REGION Network 15: Start dosilanie minuty
   RUNG wire#powerrail
      "Detection_Changes_Data_Word_USInt"("tempdbHold_SendingTCP.sterowanie." := "tempdbHold_SendingTCP".Start_dosilanie_1.MINUTE, "DB10_instance_SCADA." := "DB10_instance_SCADA".actDTL_RechargingOn.MINUTE, memRisingTriger_Data_ := "memRisingTriger_Data_14", "dbHold_Sending.data.stat.control." := "dbHold_Sending".data."Time".Start_dosilanie_1.MINUTE)
      "Saving_Canged_Data_Word_USInt"("dbHold_download.sterowanie" := "dbHold_download".SendingTimes.Start_dosilanie_1.MINUTE, "DB10_instance_SCADA." := "DB10_instance_SCADA".actDTL_RechargingOn.MINUTE, memTrig_Client_Receiving_ := "memTrig_Client_Receiving_14")
   END_RUNG
   // the same network as SCL:
   "Detection_Changes_Data_Word_USInt"("tempdbHold_SendingTCP.sterowanie." := "tempdbHold_SendingTCP".Start_dosilanie_1.MINUTE,
                           "DB10_instance_SCADA." := "DB10_instance_SCADA".actDTL_RechargingOn.MINUTE,
                           memRisingTriger_Data_ := "memRisingTriger_Data_14",
                           "dbHold_Sending.data.stat.control." := "dbHold_Sending".data."Time".Start_dosilanie_1.MINUTE,
                           ENO => #_w1);
   IF #_w1 THEN
       "Saving_Canged_Data_Word_USInt"("dbHold_download.sterowanie" := "dbHold_download".SendingTimes.Start_dosilanie_1.MINUTE,
                               "DB10_instance_SCADA." := "DB10_instance_SCADA".actDTL_RechargingOn.MINUTE,
                               memTrig_Client_Receiving_ := "memTrig_Client_Receiving_14");
   END_IF;
END_REGION

REGION Network 16: Stop dosilanie godziny
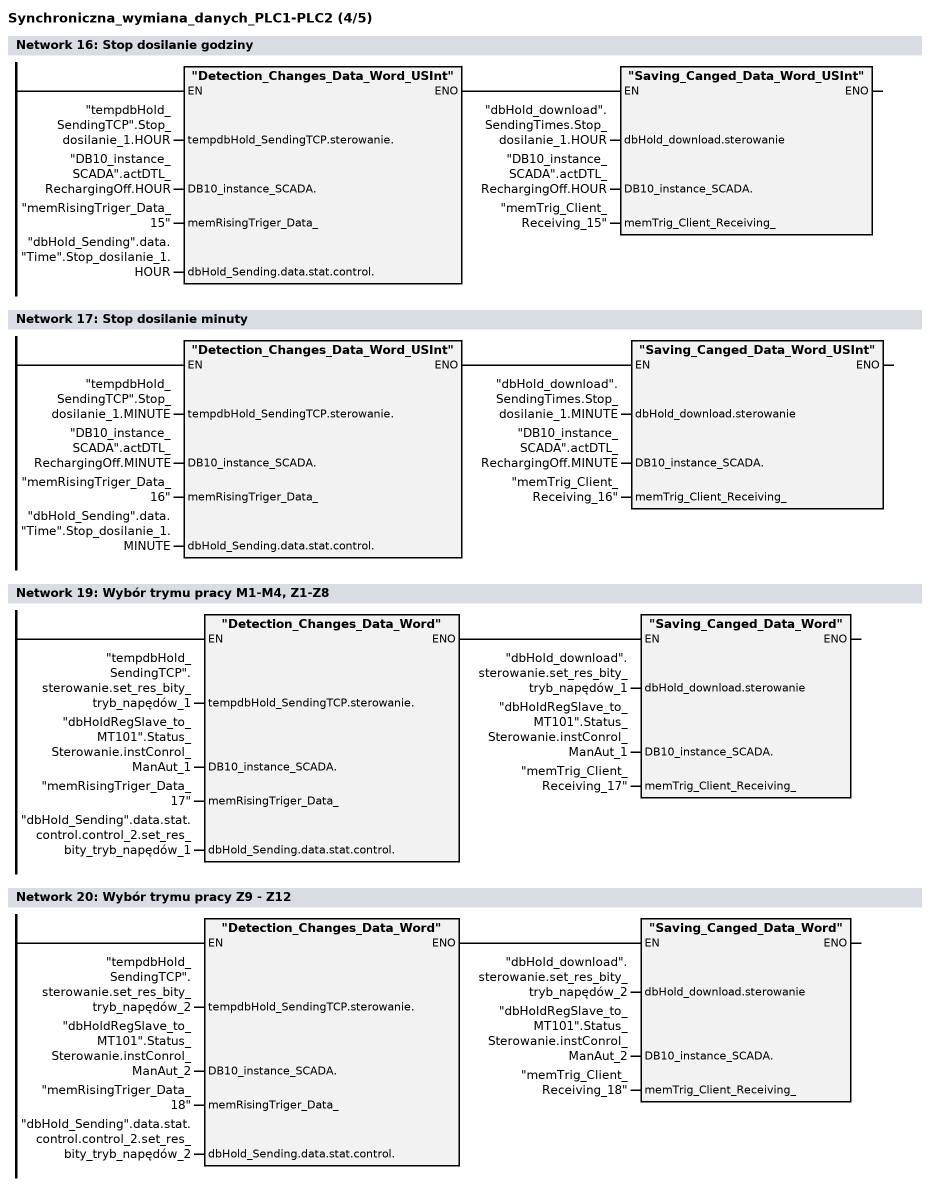
   RUNG wire#powerrail
      "Detection_Changes_Data_Word_USInt"("tempdbHold_SendingTCP.sterowanie." := "tempdbHold_SendingTCP".Stop_dosilanie_1.HOUR, "DB10_instance_SCADA." := "DB10_instance_SCADA".actDTL_RechargingOff.HOUR, memRisingTriger_Data_ := "memRisingTriger_Data_15", "dbHold_Sending.data.stat.control." := "dbHold_Sending".data."Time".Stop_dosilanie_1.HOUR)
      "Saving_Canged_Data_Word_USInt"("dbHold_download.sterowanie" := "dbHold_download".SendingTimes.Stop_dosilanie_1.HOUR, "DB10_instance_SCADA." := "DB10_instance_SCADA".actDTL_RechargingOff.HOUR, memTrig_Client_Receiving_ := "memTrig_Client_Receiving_15")
   END_RUNG
   // the same network as SCL:
   "Detection_Changes_Data_Word_USInt"("tempdbHold_SendingTCP.sterowanie." := "tempdbHold_SendingTCP".Stop_dosilanie_1.HOUR,
                           "DB10_instance_SCADA." := "DB10_instance_SCADA".actDTL_RechargingOff.HOUR,
                           memRisingTriger_Data_ := "memRisingTriger_Data_15",
                           "dbHold_Sending.data.stat.control." := "dbHold_Sending".data."Time".Stop_dosilanie_1.HOUR,
                           ENO => #_w1);
   IF #_w1 THEN
       "Saving_Canged_Data_Word_USInt"("dbHold_download.sterowanie" := "dbHold_download".SendingTimes.Stop_dosilanie_1.HOUR,
                               "DB10_instance_SCADA." := "DB10_instance_SCADA".actDTL_RechargingOff.HOUR,
                               memTrig_Client_Receiving_ := "memTrig_Client_Receiving_15");
   END_IF;
END_REGION

REGION Network 17: Stop dosilanie minuty
   RUNG wire#powerrail
      "Detection_Changes_Data_Word_USInt"("tempdbHold_SendingTCP.sterowanie." := "tempdbHold_SendingTCP".Stop_dosilanie_1.MINUTE, "DB10_instance_SCADA." := "DB10_instance_SCADA".actDTL_RechargingOff.MINUTE, memRisingTriger_Data_ := "memRisingTriger_Data_16", "dbHold_Sending.data.stat.control." := "dbHold_Sending".data."Time".Stop_dosilanie_1.MINUTE)
      "Saving_Canged_Data_Word_USInt"("dbHold_download.sterowanie" := "dbHold_download".SendingTimes.Stop_dosilanie_1.MINUTE, "DB10_instance_SCADA." := "DB10_instance_SCADA".actDTL_RechargingOff.MINUTE, memTrig_Client_Receiving_ := "memTrig_Client_Receiving_16")
   END_RUNG
   // the same network as SCL:
   "Detection_Changes_Data_Word_USInt"("tempdbHold_SendingTCP.sterowanie." := "tempdbHold_SendingTCP".Stop_dosilanie_1.MINUTE,
                           "DB10_instance_SCADA." := "DB10_instance_SCADA".actDTL_RechargingOff.MINUTE,
                           memRisingTriger_Data_ := "memRisingTriger_Data_16",
                           "dbHold_Sending.data.stat.control." := "dbHold_Sending".data."Time".Stop_dosilanie_1.MINUTE,
                           ENO => #_w1);
   IF #_w1 THEN
       "Saving_Canged_Data_Word_USInt"("dbHold_download.sterowanie" := "dbHold_download".SendingTimes.Stop_dosilanie_1.MINUTE,
                               "DB10_instance_SCADA." := "DB10_instance_SCADA".actDTL_RechargingOff.MINUTE,
                               memTrig_Client_Receiving_ := "memTrig_Client_Receiving_16");
   END_IF;
END_REGION

REGION Network 19: Wybór trymu pracy M1-M4, Z1-Z8
   RUNG wire#powerrail
      "Detection_Changes_Data_Word"("tempdbHold_SendingTCP.sterowanie." := "tempdbHold_SendingTCP".sterowanie.set_res_bity_tryb_napędów_1, "DB10_instance_SCADA." := "dbHoldRegSlave_to_MT101".Status_Sterowanie.instConrol_ManAut_1, memRisingTriger_Data_ := "memRisingTriger_Data_17", "dbHold_Sending.data.stat.control." := "dbHold_Sending".data.stat.control.control_2.set_res_bity_tryb_napędów_1)
      "Saving_Canged_Data_Word"("dbHold_download.sterowanie" := "dbHold_download".sterowanie.set_res_bity_tryb_napędów_1, "DB10_instance_SCADA." := "dbHoldRegSlave_to_MT101".Status_Sterowanie.instConrol_ManAut_1, memTrig_Client_Receiving_ := "memTrig_Client_Receiving_17")
   END_RUNG
   // the same network as SCL:
   "Detection_Changes_Data_Word"("tempdbHold_SendingTCP.sterowanie." := "tempdbHold_SendingTCP".sterowanie.set_res_bity_tryb_napędów_1,
                           "DB10_instance_SCADA." := "dbHoldRegSlave_to_MT101".Status_Sterowanie.instConrol_ManAut_1,
                           memRisingTriger_Data_ := "memRisingTriger_Data_17",
                           "dbHold_Sending.data.stat.control." := "dbHold_Sending".data.stat.control.control_2.set_res_bity_tryb_napędów_1,
                           ENO => #_w1);
   IF #_w1 THEN
       "Saving_Canged_Data_Word"("dbHold_download.sterowanie" := "dbHold_download".sterowanie.set_res_bity_tryb_napędów_1,
                               "DB10_instance_SCADA." := "dbHoldRegSlave_to_MT101".Status_Sterowanie.instConrol_ManAut_1,
                               memTrig_Client_Receiving_ := "memTrig_Client_Receiving_17");
   END_IF;
END_REGION

REGION Network 20: Wybór trymu pracy Z9 - Z12
   RUNG wire#powerrail
      "Detection_Changes_Data_Word"("tempdbHold_SendingTCP.sterowanie." := "tempdbHold_SendingTCP".sterowanie.set_res_bity_tryb_napędów_2, "DB10_instance_SCADA." := "dbHoldRegSlave_to_MT101".Status_Sterowanie.instConrol_ManAut_2, memRisingTriger_Data_ := "memRisingTriger_Data_18", "dbHold_Sending.data.stat.control." := "dbHold_Sending".data.stat.control.control_2.set_res_bity_tryb_napędów_2)
      "Saving_Canged_Data_Word"("dbHold_download.sterowanie" := "dbHold_download".sterowanie.set_res_bity_tryb_napędów_2, "DB10_instance_SCADA." := "dbHoldRegSlave_to_MT101".Status_Sterowanie.instConrol_ManAut_2, memTrig_Client_Receiving_ := "memTrig_Client_Receiving_18")
   END_RUNG
   // the same network as SCL:
   "Detection_Changes_Data_Word"("tempdbHold_SendingTCP.sterowanie." := "tempdbHold_SendingTCP".sterowanie.set_res_bity_tryb_napędów_2,
                           "DB10_instance_SCADA." := "dbHoldRegSlave_to_MT101".Status_Sterowanie.instConrol_ManAut_2,
                           memRisingTriger_Data_ := "memRisingTriger_Data_18",
                           "dbHold_Sending.data.stat.control." := "dbHold_Sending".data.stat.control.control_2.set_res_bity_tryb_napędów_2,
                           ENO => #_w1);
   IF #_w1 THEN
       "Saving_Canged_Data_Word"("dbHold_download.sterowanie" := "dbHold_download".sterowanie.set_res_bity_tryb_napędów_2,
                               "DB10_instance_SCADA." := "dbHoldRegSlave_to_MT101".Status_Sterowanie.instConrol_ManAut_2,
                               memTrig_Client_Receiving_ := "memTrig_Client_Receiving_18");
   END_IF;
END_REGION

REGION Network 21: Sterowanie OTWIERANIE/ZAMYKANIE Z1 - Z8
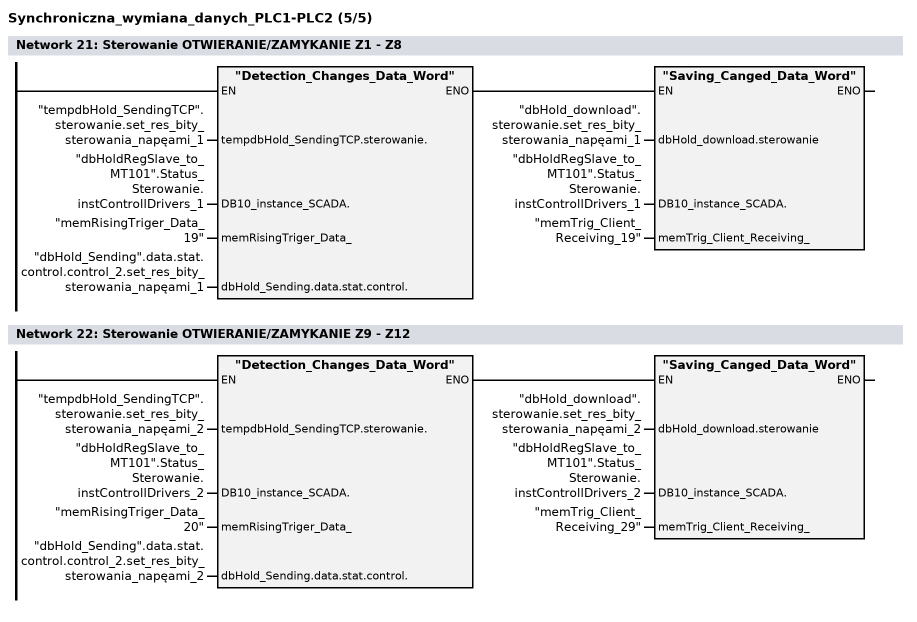
   RUNG wire#powerrail
      "Detection_Changes_Data_Word"("tempdbHold_SendingTCP.sterowanie." := "tempdbHold_SendingTCP".sterowanie.set_res_bity_sterowania_napęami_1, "DB10_instance_SCADA." := "dbHoldRegSlave_to_MT101".Status_Sterowanie.instControllDrivers_1, memRisingTriger_Data_ := "memRisingTriger_Data_19", "dbHold_Sending.data.stat.control." := "dbHold_Sending".data.stat.control.control_2.set_res_bity_sterowania_napęami_1)
      "Saving_Canged_Data_Word"("dbHold_download.sterowanie" := "dbHold_download".sterowanie.set_res_bity_sterowania_napęami_1, "DB10_instance_SCADA." := "dbHoldRegSlave_to_MT101".Status_Sterowanie.instControllDrivers_1, memTrig_Client_Receiving_ := "memTrig_Client_Receiving_19")
   END_RUNG
   // the same network as SCL:
   "Detection_Changes_Data_Word"("tempdbHold_SendingTCP.sterowanie." := "tempdbHold_SendingTCP".sterowanie.set_res_bity_sterowania_napęami_1,
                           "DB10_instance_SCADA." := "dbHoldRegSlave_to_MT101".Status_Sterowanie.instControllDrivers_1,
                           memRisingTriger_Data_ := "memRisingTriger_Data_19",
                           "dbHold_Sending.data.stat.control." := "dbHold_Sending".data.stat.control.control_2.set_res_bity_sterowania_napęami_1,
                           ENO => #_w1);
   IF #_w1 THEN
       "Saving_Canged_Data_Word"("dbHold_download.sterowanie" := "dbHold_download".sterowanie.set_res_bity_sterowania_napęami_1,
                               "DB10_instance_SCADA." := "dbHoldRegSlave_to_MT101".Status_Sterowanie.instControllDrivers_1,
                               memTrig_Client_Receiving_ := "memTrig_Client_Receiving_19");
   END_IF;
END_REGION

REGION Network 22: Sterowanie OTWIERANIE/ZAMYKANIE Z9 - Z12
   RUNG wire#powerrail
      "Detection_Changes_Data_Word"("tempdbHold_SendingTCP.sterowanie." := "tempdbHold_SendingTCP".sterowanie.set_res_bity_sterowania_napęami_2, "DB10_instance_SCADA." := "dbHoldRegSlave_to_MT101".Status_Sterowanie.instControllDrivers_2, memRisingTriger_Data_ := "memRisingTriger_Data_20", "dbHold_Sending.data.stat.control." := "dbHold_Sending".data.stat.control.control_2.set_res_bity_sterowania_napęami_2)
      "Saving_Canged_Data_Word"("dbHold_download.sterowanie" := "dbHold_download".sterowanie.set_res_bity_sterowania_napęami_2, "DB10_instance_SCADA." := "dbHoldRegSlave_to_MT101".Status_Sterowanie.instControllDrivers_2, memTrig_Client_Receiving_ := "memTrig_Client_Receiving_29")
   END_RUNG
   // the same network as SCL:
   "Detection_Changes_Data_Word"("tempdbHold_SendingTCP.sterowanie." := "tempdbHold_SendingTCP".sterowanie.set_res_bity_sterowania_napęami_2,
                           "DB10_instance_SCADA." := "dbHoldRegSlave_to_MT101".Status_Sterowanie.instControllDrivers_2,
                           memRisingTriger_Data_ := "memRisingTriger_Data_20",
                           "dbHold_Sending.data.stat.control." := "dbHold_Sending".data.stat.control.control_2.set_res_bity_sterowania_napęami_2,
                           ENO => #_w1);
   IF #_w1 THEN
       "Saving_Canged_Data_Word"("dbHold_download.sterowanie" := "dbHold_download".sterowanie.set_res_bity_sterowania_napęami_2,
                               "DB10_instance_SCADA." := "dbHoldRegSlave_to_MT101".Status_Sterowanie.instControllDrivers_2,
                               memTrig_Client_Receiving_ := "memTrig_Client_Receiving_29");
   END_IF;
END_REGION
END_FUNCTION

FUNCTION "Detection_Changes_Data_Real" : Void   // FC33, LAD
{ S7_Optimized_Access := 'TRUE' }
AUTHOR : rtecmer
VERSION : 0.1
// Funkcja porównuje wartości w bloku wymiany danych i jeśli zaszła zmiana wprowadza ją
// stored: AutoNumber true, IsIECCheckEnabled false, SetENOAutomatically false, UDAEnableTagReadback false
   VAR_IN_OUT
      "tempdbHold_SendingTCP.sterowanie." : Real;   // zadana wartośc zmiennej do porównania
      "DB10_instance_SCADA." : Real;   // zmienna w db której porównujemy
      memRisingTriger_Data_ : Bool;   // bit pamięci zbocza zmiany
      "dbHold_Sending.data.stat.control." : Real;   // zmienna w db wyjścia do zmiany
   END_VAR
   VAR_TEMP   // added for the SCL form of the ladder/FBD networks
      _w1 : Bool;
      _w2 : Bool;
   END_VAR
BEGIN

REGION Network 1: bit inicjacji wysłąnia nowej wartości
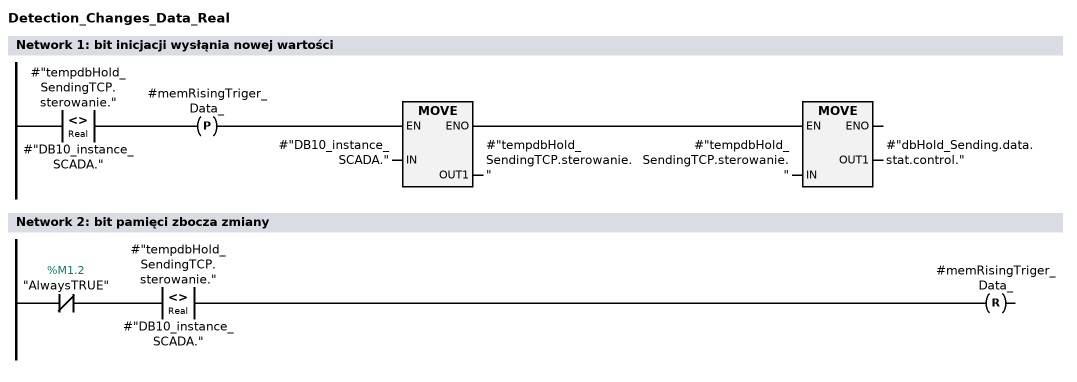
   RUNG wire#powerrail
      { S7_Templates := "SrcType := Real" } NE_Contact(in1 := #"tempdbHold_SendingTCP.sterowanie.", in2 := #"DB10_instance_SCADA.")
      P_Trig( #memRisingTriger_Data_ )
      Move(in := #"DB10_instance_SCADA.", out1 => #"tempdbHold_SendingTCP.sterowanie.")
      Move(in := #"tempdbHold_SendingTCP.sterowanie.", out1 => #"dbHold_Sending.data.stat.control.")
   END_RUNG
   // the same network as SCL:
   #_w1 := #"tempdbHold_SendingTCP.sterowanie." <> #"DB10_instance_SCADA.";
   #_w2 := #_w1 AND NOT #memRisingTriger_Data_;   // rising edge
   #memRisingTriger_Data_ := #_w1;
   IF #_w2 THEN
       #"tempdbHold_SendingTCP.sterowanie." := #"DB10_instance_SCADA.";
       #"dbHold_Sending.data.stat.control." := #"tempdbHold_SendingTCP.sterowanie.";
   END_IF;
END_REGION

REGION Network 2: bit pamięci zbocza zmiany
   RUNG wire#powerrail
      I_Contact( "AlwaysTRUE" )
      { S7_Templates := "SrcType := Real" } NE_Contact(in1 := #"tempdbHold_SendingTCP.sterowanie.", in2 := #"DB10_instance_SCADA.")
      R_Coil( #memRisingTriger_Data_ )
   END_RUNG
   // the same network as SCL:
   IF NOT "AlwaysTRUE" AND (#"tempdbHold_SendingTCP.sterowanie." <> #"DB10_instance_SCADA.") THEN
       #memRisingTriger_Data_ := FALSE;
   END_IF;
END_REGION
END_FUNCTION

FUNCTION "Saving_Canged_Data_Real" : Void   // FC32, LAD
{ S7_Optimized_Access := 'TRUE' }
AUTHOR : rtecmer
VERSION : 0.1
// Funkcj po sprawdzeniu czy dane w pobranym bloku różnią się od danyc w bloku SCADA dokonuje operacji zapisu jeśli byatąpiła różnica danych.
// stored: AutoNumber true, IsIECCheckEnabled false, SetENOAutomatically false, UDAEnableTagReadback false
   VAR_IN_OUT
      "dbHold_download.sterowanie" : Real;   // Zmienna zadawana i porównywana
      "DB10_instance_SCADA." : Real;   // Zmienna do porównania
      memTrig_Client_Receiving_ : Bool;   // pamięć zbocze zmiany
   END_VAR
   VAR_TEMP   // added for the SCL form of the ladder/FBD networks
      _w1 : Bool;
      _w2 : Bool;
   END_VAR
BEGIN

REGION Network 1
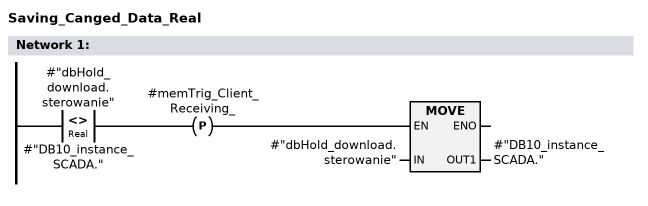
   RUNG wire#powerrail
      { S7_Templates := "SrcType := Real" } NE_Contact(in1 := #"dbHold_download.sterowanie", in2 := #"DB10_instance_SCADA.")
      P_Trig( #memTrig_Client_Receiving_ )
      Move(in := #"dbHold_download.sterowanie", out1 => #"DB10_instance_SCADA.")
   END_RUNG
   // the same network as SCL:
   #_w1 := #"dbHold_download.sterowanie" <> #"DB10_instance_SCADA.";
   #_w2 := #_w1 AND NOT #memTrig_Client_Receiving_;   // rising edge
   #memTrig_Client_Receiving_ := #_w1;
   IF #_w2 THEN #"DB10_instance_SCADA." := #"dbHold_download.sterowanie"; END_IF;
END_REGION
END_FUNCTION

FUNCTION "Detection_Changes_Data_Word" : Void   // FC35, LAD
{ S7_Optimized_Access := 'TRUE' }
AUTHOR : rtecmer
VERSION : 0.1
// Funkcja porównuje wartości w bloku wymiany danych i jeśli zaszła zmiana wprowadza ją
// stored: AutoNumber false, IsIECCheckEnabled false, SetENOAutomatically false, UDAEnableTagReadback false
   VAR_IN_OUT
      "tempdbHold_SendingTCP.sterowanie." : Int;   // zadana wartośc zmiennej do porównania
      "DB10_instance_SCADA." : Int;   // zmienna w db której porównujemy
      memRisingTriger_Data_ : Bool;   // bit pamięci zbocza zmiany
      "dbHold_Sending.data.stat.control." : Int;   // zmienna w db wyjścia do zmiany
   END_VAR
   VAR_TEMP   // added for the SCL form of the ladder/FBD networks
      _w1 : Bool;
      _w2 : Bool;
   END_VAR
BEGIN

REGION Network 1: bit inicjacji wysłąnia nowej wartości
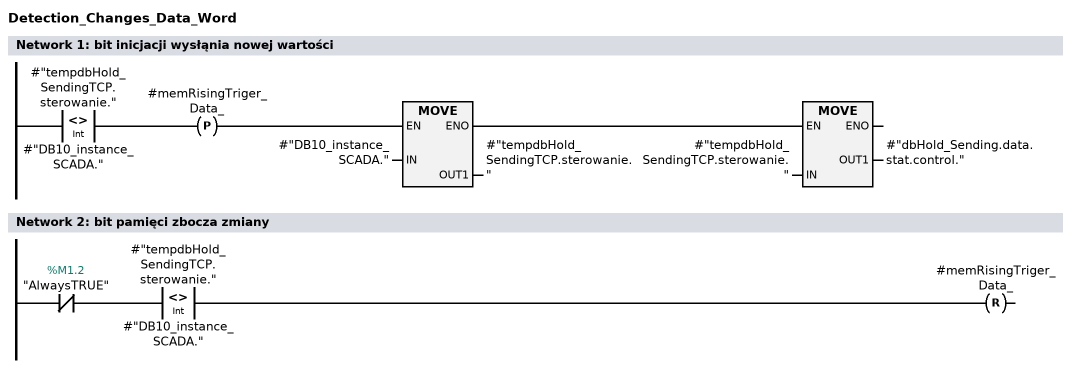
   RUNG wire#powerrail
      { S7_Templates := "SrcType := Int" } NE_Contact(in1 := #"tempdbHold_SendingTCP.sterowanie.", in2 := #"DB10_instance_SCADA.")
      P_Trig( #memRisingTriger_Data_ )
      Move(in := #"DB10_instance_SCADA.", out1 => #"tempdbHold_SendingTCP.sterowanie.")
      Move(in := #"tempdbHold_SendingTCP.sterowanie.", out1 => #"dbHold_Sending.data.stat.control.")
   END_RUNG
   // the same network as SCL:
   #_w1 := #"tempdbHold_SendingTCP.sterowanie." <> #"DB10_instance_SCADA.";
   #_w2 := #_w1 AND NOT #memRisingTriger_Data_;   // rising edge
   #memRisingTriger_Data_ := #_w1;
   IF #_w2 THEN
       #"tempdbHold_SendingTCP.sterowanie." := #"DB10_instance_SCADA.";
       #"dbHold_Sending.data.stat.control." := #"tempdbHold_SendingTCP.sterowanie.";
   END_IF;
END_REGION

REGION Network 2: bit pamięci zbocza zmiany
   RUNG wire#powerrail
      I_Contact( "AlwaysTRUE" )
      { S7_Templates := "SrcType := Int" } NE_Contact(in1 := #"tempdbHold_SendingTCP.sterowanie.", in2 := #"DB10_instance_SCADA.")
      R_Coil( #memRisingTriger_Data_ )
   END_RUNG
   // the same network as SCL:
   IF NOT "AlwaysTRUE" AND (#"tempdbHold_SendingTCP.sterowanie." <> #"DB10_instance_SCADA.") THEN
       #memRisingTriger_Data_ := FALSE;
   END_IF;
END_REGION
END_FUNCTION

FUNCTION "Saving_Canged_Data_Word" : Void   // FC36, LAD
{ S7_Optimized_Access := 'TRUE' }
AUTHOR : rtecmer
VERSION : 0.1
// Funkcj po sprawdzeniu czy dane w pobranym bloku różnią się od danyc w bloku SCADA dokonuje operacji zapisu jeśli byatąpiła różnica danych.
// stored: AutoNumber false, IsIECCheckEnabled false, SetENOAutomatically false, UDAEnableTagReadback false
   VAR_IN_OUT
      "dbHold_download.sterowanie" : Int;   // Zmienna zadawana i porównywana
      "DB10_instance_SCADA." : Int;   // Zmienna do porównania
      memTrig_Client_Receiving_ : Bool;   // pamięć zbocze zmiany
   END_VAR
   VAR_TEMP   // added for the SCL form of the ladder/FBD networks
      _w1 : Bool;
      _w2 : Bool;
   END_VAR
BEGIN

REGION Network 1
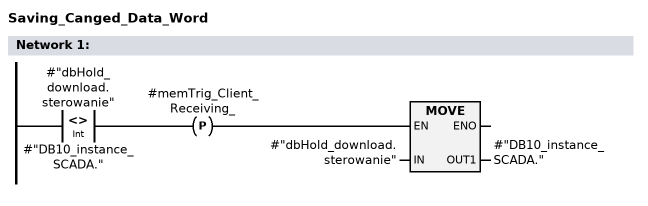
   RUNG wire#powerrail
      { S7_Templates := "SrcType := Int" } NE_Contact(in1 := #"dbHold_download.sterowanie", in2 := #"DB10_instance_SCADA.")
      P_Trig( #memTrig_Client_Receiving_ )
      Move(in := #"dbHold_download.sterowanie", out1 => #"DB10_instance_SCADA.")
   END_RUNG
   // the same network as SCL:
   #_w1 := #"dbHold_download.sterowanie" <> #"DB10_instance_SCADA.";
   #_w2 := #_w1 AND NOT #memTrig_Client_Receiving_;   // rising edge
   #memTrig_Client_Receiving_ := #_w1;
   IF #_w2 THEN #"DB10_instance_SCADA." := #"dbHold_download.sterowanie"; END_IF;
END_REGION
END_FUNCTION

FUNCTION "Detection_Changes_Data_Word_USInt" : Void   // FC37, LAD
{ S7_Optimized_Access := 'TRUE' }
AUTHOR : rtecmer
VERSION : 0.1
// Funkcja porównuje wartości w bloku wymiany danych i jeśli zaszła zmiana wprowadza ją
// stored: AutoNumber false, IsIECCheckEnabled false, SetENOAutomatically false, UDAEnableTagReadback false
   VAR_IN_OUT
      "tempdbHold_SendingTCP.sterowanie." : USInt;   // zadana wartośc zmiennej do porównania
      "DB10_instance_SCADA." : USInt;   // zmienna w db której porównujemy
      memRisingTriger_Data_ : Bool;   // bit pamięci zbocza zmiany
      "dbHold_Sending.data.stat.control." : USInt;   // zmienna w db wyjścia do zmiany
   END_VAR
   VAR_TEMP   // added for the SCL form of the ladder/FBD networks
      _w1 : Bool;
      _w2 : Bool;
   END_VAR
BEGIN

REGION Network 2: bit inicjacji wysłąnia nowej wartości
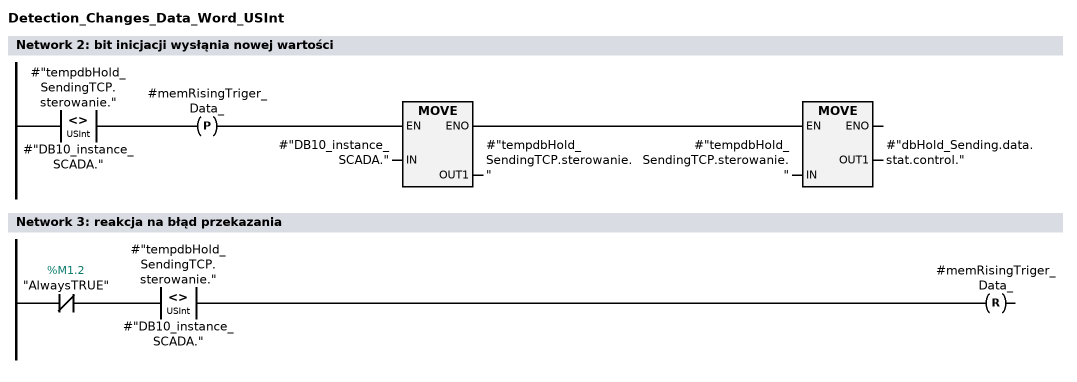
   RUNG wire#powerrail
      { S7_Templates := "SrcType := USInt" } NE_Contact(in1 := #"tempdbHold_SendingTCP.sterowanie.", in2 := #"DB10_instance_SCADA.")
      P_Trig( #memRisingTriger_Data_ )
      Move(in := #"DB10_instance_SCADA.", out1 => #"tempdbHold_SendingTCP.sterowanie.")
      Move(in := #"tempdbHold_SendingTCP.sterowanie.", out1 => #"dbHold_Sending.data.stat.control.")
   END_RUNG
   // the same network as SCL:
   #_w1 := #"tempdbHold_SendingTCP.sterowanie." <> #"DB10_instance_SCADA.";
   #_w2 := #_w1 AND NOT #memRisingTriger_Data_;   // rising edge
   #memRisingTriger_Data_ := #_w1;
   IF #_w2 THEN
       #"tempdbHold_SendingTCP.sterowanie." := #"DB10_instance_SCADA.";
       #"dbHold_Sending.data.stat.control." := #"tempdbHold_SendingTCP.sterowanie.";
   END_IF;
END_REGION

REGION Network 3: reakcja na błąd przekazania
   RUNG wire#powerrail
      I_Contact( "AlwaysTRUE" )
      { S7_Templates := "SrcType := USInt" } NE_Contact(in1 := #"tempdbHold_SendingTCP.sterowanie.", in2 := #"DB10_instance_SCADA.")
      R_Coil( #memRisingTriger_Data_ )
   END_RUNG
   // the same network as SCL:
   IF NOT "AlwaysTRUE" AND (#"tempdbHold_SendingTCP.sterowanie." <> #"DB10_instance_SCADA.") THEN
       #memRisingTriger_Data_ := FALSE;
   END_IF;
END_REGION
END_FUNCTION

FUNCTION "Saving_Canged_Data_Word_USInt" : Void   // FC38, LAD
{ S7_Optimized_Access := 'TRUE' }
AUTHOR : rtecmer
VERSION : 0.1
// Funkcj po sprawdzeniu czy dane w pobranym bloku różnią się od danyc w bloku SCADA dokonuje operacji zapisu jeśli byatąpiła różnica danych.
// stored: AutoNumber false, IsIECCheckEnabled false, SetENOAutomatically false, UDAEnableTagReadback false
   VAR_IN_OUT
      "dbHold_download.sterowanie" : USInt;   // Zmienna zadawana i porównywana
      "DB10_instance_SCADA." : USInt;   // Zmienna do porównania
      memTrig_Client_Receiving_ : Bool;   // pamięć zbocze zmiany
   END_VAR
   VAR_TEMP
      dbHold_download : Int;
   END_VAR
   VAR_TEMP   // added for the SCL form of the ladder/FBD networks
      _w1 : Bool;
      _w2 : Bool;
   END_VAR
BEGIN

REGION Network 2
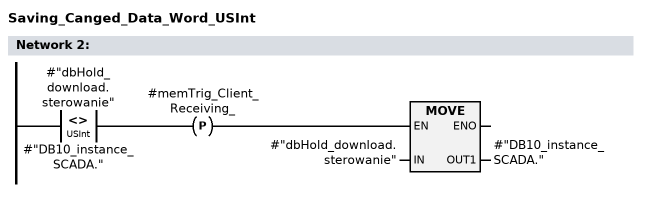
   RUNG wire#powerrail
      { S7_Templates := "SrcType := USInt" } NE_Contact(in1 := #"dbHold_download.sterowanie", in2 := #"DB10_instance_SCADA.")
      P_Trig( #memTrig_Client_Receiving_ )
      Move(in := #"dbHold_download.sterowanie", out1 => #"DB10_instance_SCADA.")
   END_RUNG
   // the same network as SCL:
   #_w1 := #"dbHold_download.sterowanie" <> #"DB10_instance_SCADA.";
   #_w2 := #_w1 AND NOT #memTrig_Client_Receiving_;   // rising edge
   #memTrig_Client_Receiving_ := #_w1;
   IF #_w2 THEN #"DB10_instance_SCADA." := #"dbHold_download.sterowanie"; END_IF;
END_REGION
END_FUNCTION

FUNCTION "Sterowniki napędów" : Void   // FC7, LAD
TITLE = Sterowniki
{ S7_Optimized_Access := 'TRUE' }
AUTHOR : rtecmer
VERSION : 0.1
// Sterownik napędów zasuw Z1-Z9
// stored: AutoNumber true, IsIECCheckEnabled false, SetENOAutomatically false, UDAEnableTagReadback false
BEGIN

REGION Network 2: Sterowanie Zasuwą Z10 - Położenie
   // Funkcja zawiera kontrolę czasu jazdy na pozycję ustawiony czas 120sek
   // po upływie czasu nastapi alarm i przełączenie w trym manual
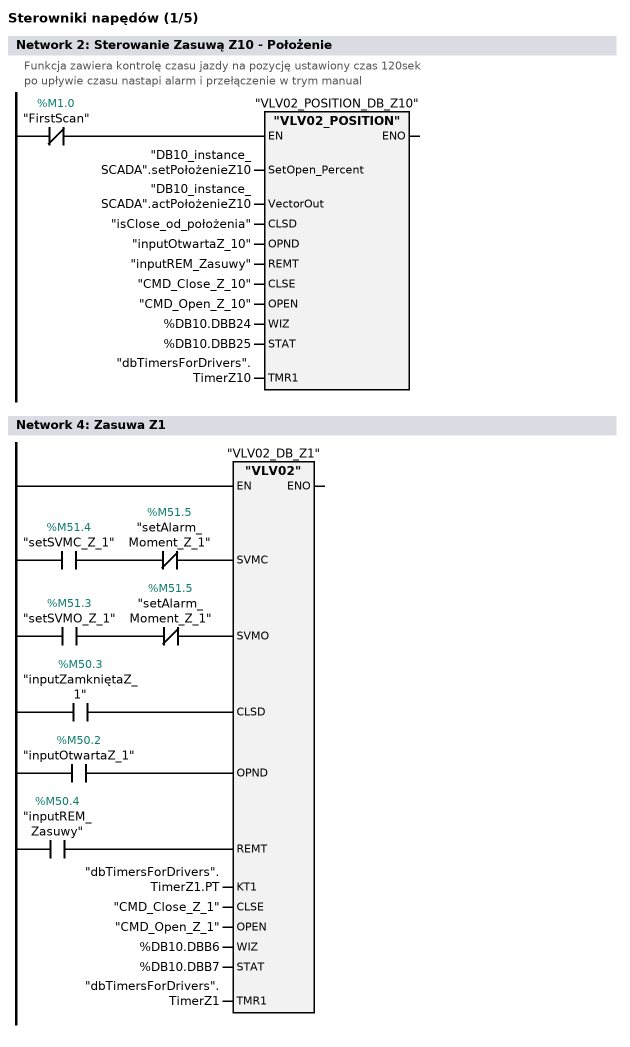
   RUNG wire#powerrail
      I_Contact( "FirstScan" )
      "VLV02_POSITION_DB_Z10"(SetOpen_Percent := "DB10_instance_SCADA".setPołożenieZ10, VectorOut := "DB10_instance_SCADA".actPołożenieZ10, CLSD := "isClose_od_położenia", OPND := "inputOtwartaZ_10", REMT := "inputREM_Zasuwy", CLSE := "CMD_Close_Z_10", OPEN := "CMD_Open_Z_10", WIZ := %DB10.DBB24, STAT := %DB10.DBB25, TMR1 := "dbTimersForDrivers".TimerZ10)
   END_RUNG
   // the same network as SCL:
   IF NOT "FirstScan" THEN
       "VLV02_POSITION_DB_Z10"(SetOpen_Percent := "DB10_instance_SCADA".setPołożenieZ10,   // "VLV02_POSITION"
                               VectorOut := "DB10_instance_SCADA".actPołożenieZ10,
                               CLSD := "isClose_od_położenia",
                               OPND := "inputOtwartaZ_10",
                               REMT := "inputREM_Zasuwy",
                               CLSE := "CMD_Close_Z_10",
                               OPEN := "CMD_Open_Z_10",
                               WIZ := %DB10.DBB24,
                               STAT := %DB10.DBB25,
                               TMR1 := "dbTimersForDrivers".TimerZ10);
   END_IF;
END_REGION

REGION Network 4: Zasuwa Z1
   RUNG wire#powerrail
      "VLV02_DB_Z1"(SVMC := wire#w1, SVMO := wire#w2, CLSD := wire#w3, OPND := wire#w4, REMT := wire#w5, KT1 := "dbTimersForDrivers".TimerZ1.PT, CLSE := "CMD_Close_Z_1", OPEN := "CMD_Open_Z_1", WIZ := %DB10.DBB6, STAT := %DB10.DBB7, TMR1 := "dbTimersForDrivers".TimerZ1)
   END_RUNG
   RUNG wire#powerrail
      Contact( "setSVMC_Z_1" )
      I_Contact( "setAlarm_Moment_Z_1" )
   END_RUNG wire#w1
   RUNG wire#powerrail
      Contact( "setSVMO_Z_1" )
      I_Contact( "setAlarm_Moment_Z_1" )
   END_RUNG wire#w2
   RUNG wire#powerrail
      Contact( "inputZamkniętaZ_1" )
   END_RUNG wire#w3
   RUNG wire#powerrail
      Contact( "inputOtwartaZ_1" )
   END_RUNG wire#w4
   RUNG wire#powerrail
      Contact( "inputREM_Zasuwy" )
   END_RUNG wire#w5
   // the same network as SCL:
   "VLV02_DB_Z1"(SVMC := "setSVMC_Z_1" AND NOT "setAlarm_Moment_Z_1",   // "VLV02"
                 SVMO := "setSVMO_Z_1" AND NOT "setAlarm_Moment_Z_1",
                 CLSD := "inputZamkniętaZ_1",
                 OPND := "inputOtwartaZ_1",
                 REMT := "inputREM_Zasuwy",
                 KT1 := "dbTimersForDrivers".TimerZ1.PT,
                 CLSE := "CMD_Close_Z_1",
                 OPEN := "CMD_Open_Z_1",
                 WIZ := %DB10.DBB6,
                 STAT := %DB10.DBB7,
                 TMR1 := "dbTimersForDrivers".TimerZ1);
END_REGION

REGION Network 5: Zasuwa Z2
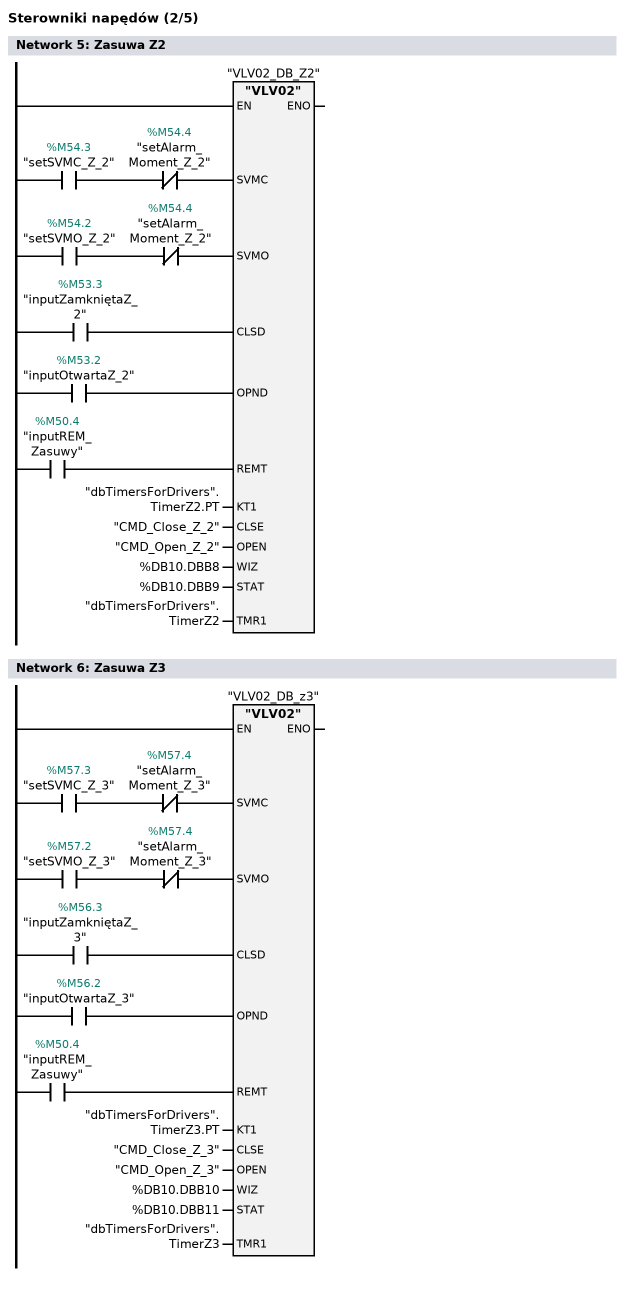
   RUNG wire#powerrail
      "VLV02_DB_Z2"(SVMC := wire#w1, SVMO := wire#w2, CLSD := wire#w3, OPND := wire#w4, REMT := wire#w5, KT1 := "dbTimersForDrivers".TimerZ2.PT, CLSE := "CMD_Close_Z_2", OPEN := "CMD_Open_Z_2", WIZ := %DB10.DBB8, STAT := %DB10.DBB9, TMR1 := "dbTimersForDrivers".TimerZ2)
   END_RUNG
   RUNG wire#powerrail
      Contact( "setSVMC_Z_2" )
      I_Contact( "setAlarm_Moment_Z_2" )
   END_RUNG wire#w1
   RUNG wire#powerrail
      Contact( "setSVMO_Z_2" )
      I_Contact( "setAlarm_Moment_Z_2" )
   END_RUNG wire#w2
   RUNG wire#powerrail
      Contact( "inputZamkniętaZ_2" )
   END_RUNG wire#w3
   RUNG wire#powerrail
      Contact( "inputOtwartaZ_2" )
   END_RUNG wire#w4
   RUNG wire#powerrail
      Contact( "inputREM_Zasuwy" )
   END_RUNG wire#w5
   // the same network as SCL:
   "VLV02_DB_Z2"(SVMC := "setSVMC_Z_2" AND NOT "setAlarm_Moment_Z_2",   // "VLV02"
                 SVMO := "setSVMO_Z_2" AND NOT "setAlarm_Moment_Z_2",
                 CLSD := "inputZamkniętaZ_2",
                 OPND := "inputOtwartaZ_2",
                 REMT := "inputREM_Zasuwy",
                 KT1 := "dbTimersForDrivers".TimerZ2.PT,
                 CLSE := "CMD_Close_Z_2",
                 OPEN := "CMD_Open_Z_2",
                 WIZ := %DB10.DBB8,
                 STAT := %DB10.DBB9,
                 TMR1 := "dbTimersForDrivers".TimerZ2);
END_REGION

REGION Network 6: Zasuwa Z3
   RUNG wire#powerrail
      "VLV02_DB_z3"(SVMC := wire#w1, SVMO := wire#w2, CLSD := wire#w3, OPND := wire#w4, REMT := wire#w5, KT1 := "dbTimersForDrivers".TimerZ3.PT, CLSE := "CMD_Close_Z_3", OPEN := "CMD_Open_Z_3", WIZ := %DB10.DBB10, STAT := %DB10.DBB11, TMR1 := "dbTimersForDrivers".TimerZ3)
   END_RUNG
   RUNG wire#powerrail
      Contact( "setSVMC_Z_3" )
      I_Contact( "setAlarm_Moment_Z_3" )
   END_RUNG wire#w1
   RUNG wire#powerrail
      Contact( "setSVMO_Z_3" )
      I_Contact( "setAlarm_Moment_Z_3" )
   END_RUNG wire#w2
   RUNG wire#powerrail
      Contact( "inputZamkniętaZ_3" )
   END_RUNG wire#w3
   RUNG wire#powerrail
      Contact( "inputOtwartaZ_3" )
   END_RUNG wire#w4
   RUNG wire#powerrail
      Contact( "inputREM_Zasuwy" )
   END_RUNG wire#w5
   // the same network as SCL:
   "VLV02_DB_z3"(SVMC := "setSVMC_Z_3" AND NOT "setAlarm_Moment_Z_3",   // "VLV02"
                 SVMO := "setSVMO_Z_3" AND NOT "setAlarm_Moment_Z_3",
                 CLSD := "inputZamkniętaZ_3",
                 OPND := "inputOtwartaZ_3",
                 REMT := "inputREM_Zasuwy",
                 KT1 := "dbTimersForDrivers".TimerZ3.PT,
                 CLSE := "CMD_Close_Z_3",
                 OPEN := "CMD_Open_Z_3",
                 WIZ := %DB10.DBB10,
                 STAT := %DB10.DBB11,
                 TMR1 := "dbTimersForDrivers".TimerZ3);
END_REGION

REGION Network 7: Zasuwa Z4
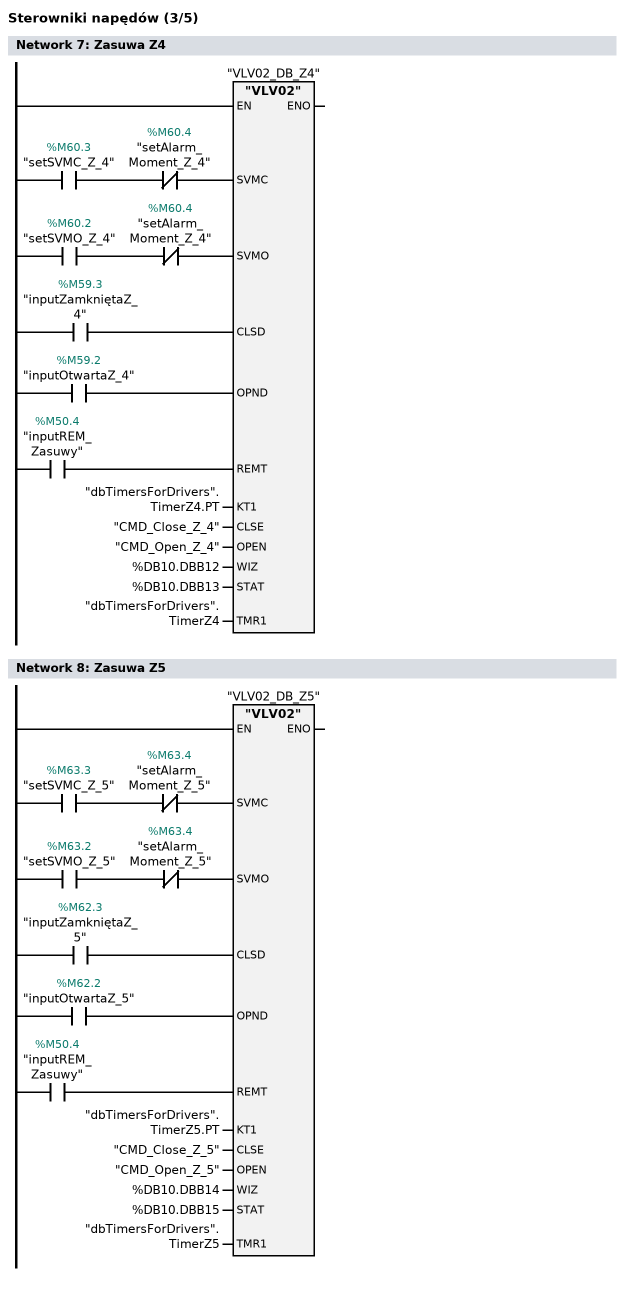
   RUNG wire#powerrail
      "VLV02_DB_Z4"(SVMC := wire#w1, SVMO := wire#w2, CLSD := wire#w3, OPND := wire#w4, REMT := wire#w5, KT1 := "dbTimersForDrivers".TimerZ4.PT, CLSE := "CMD_Close_Z_4", OPEN := "CMD_Open_Z_4", WIZ := %DB10.DBB12, STAT := %DB10.DBB13, TMR1 := "dbTimersForDrivers".TimerZ4)
   END_RUNG
   RUNG wire#powerrail
      Contact( "setSVMC_Z_4" )
      I_Contact( "setAlarm_Moment_Z_4" )
   END_RUNG wire#w1
   RUNG wire#powerrail
      Contact( "setSVMO_Z_4" )
      I_Contact( "setAlarm_Moment_Z_4" )
   END_RUNG wire#w2
   RUNG wire#powerrail
      Contact( "inputZamkniętaZ_4" )
   END_RUNG wire#w3
   RUNG wire#powerrail
      Contact( "inputOtwartaZ_4" )
   END_RUNG wire#w4
   RUNG wire#powerrail
      Contact( "inputREM_Zasuwy" )
   END_RUNG wire#w5
   // the same network as SCL:
   "VLV02_DB_Z4"(SVMC := "setSVMC_Z_4" AND NOT "setAlarm_Moment_Z_4",   // "VLV02"
                 SVMO := "setSVMO_Z_4" AND NOT "setAlarm_Moment_Z_4",
                 CLSD := "inputZamkniętaZ_4",
                 OPND := "inputOtwartaZ_4",
                 REMT := "inputREM_Zasuwy",
                 KT1 := "dbTimersForDrivers".TimerZ4.PT,
                 CLSE := "CMD_Close_Z_4",
                 OPEN := "CMD_Open_Z_4",
                 WIZ := %DB10.DBB12,
                 STAT := %DB10.DBB13,
                 TMR1 := "dbTimersForDrivers".TimerZ4);
END_REGION

REGION Network 8: Zasuwa Z5
   RUNG wire#powerrail
      "VLV02_DB_Z5"(SVMC := wire#w1, SVMO := wire#w2, CLSD := wire#w3, OPND := wire#w4, REMT := wire#w5, KT1 := "dbTimersForDrivers".TimerZ5.PT, CLSE := "CMD_Close_Z_5", OPEN := "CMD_Open_Z_5", WIZ := %DB10.DBB14, STAT := %DB10.DBB15, TMR1 := "dbTimersForDrivers".TimerZ5)
   END_RUNG
   RUNG wire#powerrail
      Contact( "setSVMC_Z_5" )
      I_Contact( "setAlarm_Moment_Z_5" )
   END_RUNG wire#w1
   RUNG wire#powerrail
      Contact( "setSVMO_Z_5" )
      I_Contact( "setAlarm_Moment_Z_5" )
   END_RUNG wire#w2
   RUNG wire#powerrail
      Contact( "inputZamkniętaZ_5" )
   END_RUNG wire#w3
   RUNG wire#powerrail
      Contact( "inputOtwartaZ_5" )
   END_RUNG wire#w4
   RUNG wire#powerrail
      Contact( "inputREM_Zasuwy" )
   END_RUNG wire#w5
   // the same network as SCL:
   "VLV02_DB_Z5"(SVMC := "setSVMC_Z_5" AND NOT "setAlarm_Moment_Z_5",   // "VLV02"
                 SVMO := "setSVMO_Z_5" AND NOT "setAlarm_Moment_Z_5",
                 CLSD := "inputZamkniętaZ_5",
                 OPND := "inputOtwartaZ_5",
                 REMT := "inputREM_Zasuwy",
                 KT1 := "dbTimersForDrivers".TimerZ5.PT,
                 CLSE := "CMD_Close_Z_5",
                 OPEN := "CMD_Open_Z_5",
                 WIZ := %DB10.DBB14,
                 STAT := %DB10.DBB15,
                 TMR1 := "dbTimersForDrivers".TimerZ5);
END_REGION

REGION Network 9: Zasuwa Z6
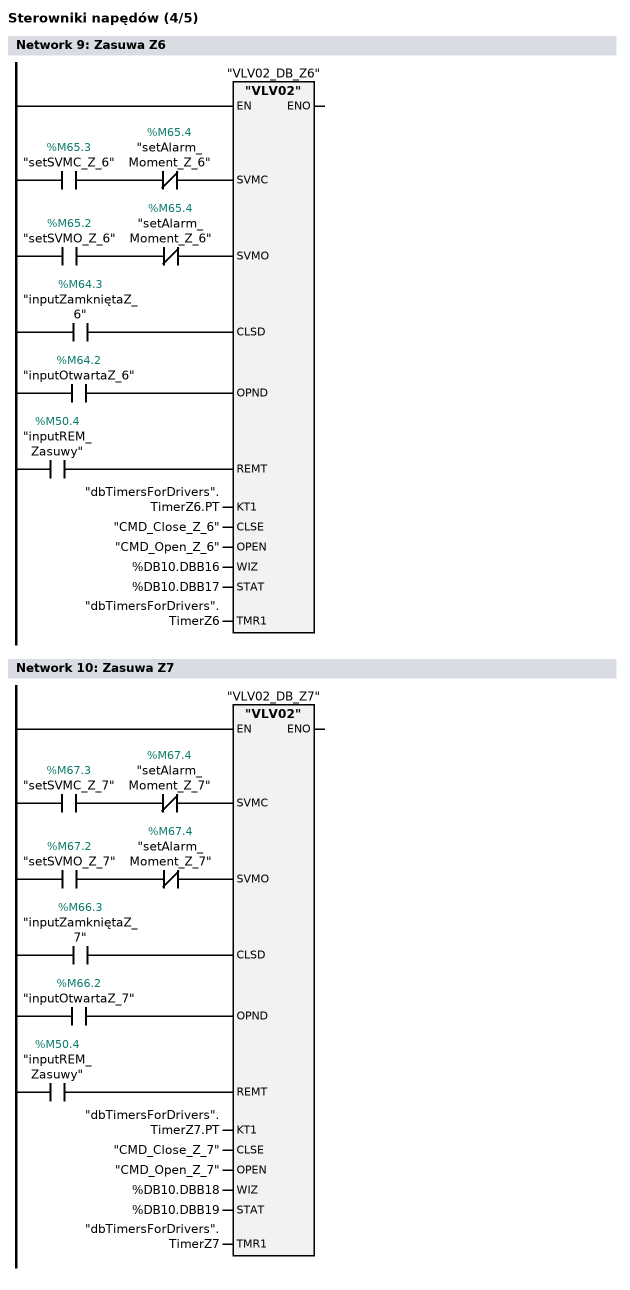
   RUNG wire#powerrail
      "VLV02_DB_Z6"(SVMC := wire#w1, SVMO := wire#w2, CLSD := wire#w3, OPND := wire#w4, REMT := wire#w5, KT1 := "dbTimersForDrivers".TimerZ6.PT, CLSE := "CMD_Close_Z_6", OPEN := "CMD_Open_Z_6", WIZ := %DB10.DBB16, STAT := %DB10.DBB17, TMR1 := "dbTimersForDrivers".TimerZ6)
   END_RUNG
   RUNG wire#powerrail
      Contact( "setSVMC_Z_6" )
      I_Contact( "setAlarm_Moment_Z_6" )
   END_RUNG wire#w1
   RUNG wire#powerrail
      Contact( "setSVMO_Z_6" )
      I_Contact( "setAlarm_Moment_Z_6" )
   END_RUNG wire#w2
   RUNG wire#powerrail
      Contact( "inputZamkniętaZ_6" )
   END_RUNG wire#w3
   RUNG wire#powerrail
      Contact( "inputOtwartaZ_6" )
   END_RUNG wire#w4
   RUNG wire#powerrail
      Contact( "inputREM_Zasuwy" )
   END_RUNG wire#w5
   // the same network as SCL:
   "VLV02_DB_Z6"(SVMC := "setSVMC_Z_6" AND NOT "setAlarm_Moment_Z_6",   // "VLV02"
                 SVMO := "setSVMO_Z_6" AND NOT "setAlarm_Moment_Z_6",
                 CLSD := "inputZamkniętaZ_6",
                 OPND := "inputOtwartaZ_6",
                 REMT := "inputREM_Zasuwy",
                 KT1 := "dbTimersForDrivers".TimerZ6.PT,
                 CLSE := "CMD_Close_Z_6",
                 OPEN := "CMD_Open_Z_6",
                 WIZ := %DB10.DBB16,
                 STAT := %DB10.DBB17,
                 TMR1 := "dbTimersForDrivers".TimerZ6);
END_REGION

REGION Network 10: Zasuwa Z7
   RUNG wire#powerrail
      "VLV02_DB_Z7"(SVMC := wire#w1, SVMO := wire#w2, CLSD := wire#w3, OPND := wire#w4, REMT := wire#w5, KT1 := "dbTimersForDrivers".TimerZ7.PT, CLSE := "CMD_Close_Z_7", OPEN := "CMD_Open_Z_7", WIZ := %DB10.DBB18, STAT := %DB10.DBB19, TMR1 := "dbTimersForDrivers".TimerZ7)
   END_RUNG
   RUNG wire#powerrail
      Contact( "setSVMC_Z_7" )
      I_Contact( "setAlarm_Moment_Z_7" )
   END_RUNG wire#w1
   RUNG wire#powerrail
      Contact( "setSVMO_Z_7" )
      I_Contact( "setAlarm_Moment_Z_7" )
   END_RUNG wire#w2
   RUNG wire#powerrail
      Contact( "inputZamkniętaZ_7" )
   END_RUNG wire#w3
   RUNG wire#powerrail
      Contact( "inputOtwartaZ_7" )
   END_RUNG wire#w4
   RUNG wire#powerrail
      Contact( "inputREM_Zasuwy" )
   END_RUNG wire#w5
   // the same network as SCL:
   "VLV02_DB_Z7"(SVMC := "setSVMC_Z_7" AND NOT "setAlarm_Moment_Z_7",   // "VLV02"
                 SVMO := "setSVMO_Z_7" AND NOT "setAlarm_Moment_Z_7",
                 CLSD := "inputZamkniętaZ_7",
                 OPND := "inputOtwartaZ_7",
                 REMT := "inputREM_Zasuwy",
                 KT1 := "dbTimersForDrivers".TimerZ7.PT,
                 CLSE := "CMD_Close_Z_7",
                 OPEN := "CMD_Open_Z_7",
                 WIZ := %DB10.DBB18,
                 STAT := %DB10.DBB19,
                 TMR1 := "dbTimersForDrivers".TimerZ7);
END_REGION

REGION Network 11: Zasuwa Z8
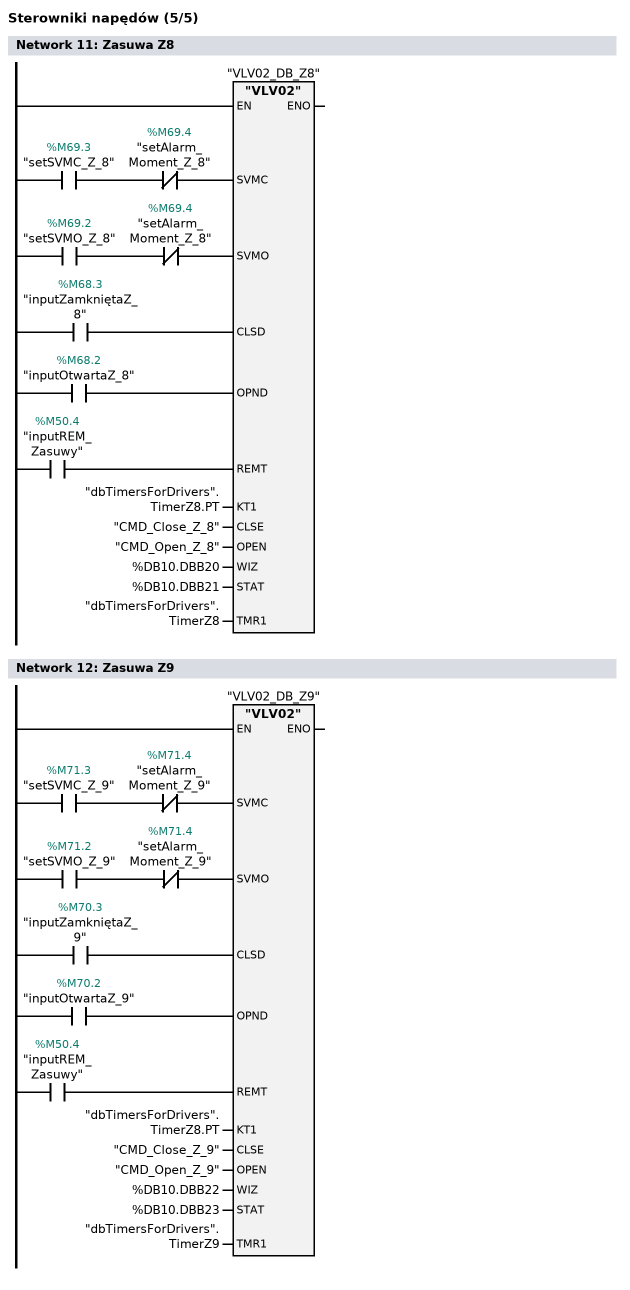
   RUNG wire#powerrail
      "VLV02_DB_Z8"(SVMC := wire#w1, SVMO := wire#w2, CLSD := wire#w3, OPND := wire#w4, REMT := wire#w5, KT1 := "dbTimersForDrivers".TimerZ8.PT, CLSE := "CMD_Close_Z_8", OPEN := "CMD_Open_Z_8", WIZ := %DB10.DBB20, STAT := %DB10.DBB21, TMR1 := "dbTimersForDrivers".TimerZ8)
   END_RUNG
   RUNG wire#powerrail
      Contact( "setSVMC_Z_8" )
      I_Contact( "setAlarm_Moment_Z_8" )
   END_RUNG wire#w1
   RUNG wire#powerrail
      Contact( "setSVMO_Z_8" )
      I_Contact( "setAlarm_Moment_Z_8" )
   END_RUNG wire#w2
   RUNG wire#powerrail
      Contact( "inputZamkniętaZ_8" )
   END_RUNG wire#w3
   RUNG wire#powerrail
      Contact( "inputOtwartaZ_8" )
   END_RUNG wire#w4
   RUNG wire#powerrail
      Contact( "inputREM_Zasuwy" )
   END_RUNG wire#w5
   // the same network as SCL:
   "VLV02_DB_Z8"(SVMC := "setSVMC_Z_8" AND NOT "setAlarm_Moment_Z_8",   // "VLV02"
                 SVMO := "setSVMO_Z_8" AND NOT "setAlarm_Moment_Z_8",
                 CLSD := "inputZamkniętaZ_8",
                 OPND := "inputOtwartaZ_8",
                 REMT := "inputREM_Zasuwy",
                 KT1 := "dbTimersForDrivers".TimerZ8.PT,
                 CLSE := "CMD_Close_Z_8",
                 OPEN := "CMD_Open_Z_8",
                 WIZ := %DB10.DBB20,
                 STAT := %DB10.DBB21,
                 TMR1 := "dbTimersForDrivers".TimerZ8);
END_REGION

REGION Network 12: Zasuwa Z9
   RUNG wire#powerrail
      "VLV02_DB_Z9"(SVMC := wire#w1, SVMO := wire#w2, CLSD := wire#w3, OPND := wire#w4, REMT := wire#w5, KT1 := "dbTimersForDrivers".TimerZ8.PT, CLSE := "CMD_Close_Z_9", OPEN := "CMD_Open_Z_9", WIZ := %DB10.DBB22, STAT := %DB10.DBB23, TMR1 := "dbTimersForDrivers".TimerZ9)
   END_RUNG
   RUNG wire#powerrail
      Contact( "setSVMC_Z_9" )
      I_Contact( "setAlarm_Moment_Z_9" )
   END_RUNG wire#w1
   RUNG wire#powerrail
      Contact( "setSVMO_Z_9" )
      I_Contact( "setAlarm_Moment_Z_9" )
   END_RUNG wire#w2
   RUNG wire#powerrail
      Contact( "inputZamkniętaZ_9" )
   END_RUNG wire#w3
   RUNG wire#powerrail
      Contact( "inputOtwartaZ_9" )
   END_RUNG wire#w4
   RUNG wire#powerrail
      Contact( "inputREM_Zasuwy" )
   END_RUNG wire#w5
   // the same network as SCL:
   "VLV02_DB_Z9"(SVMC := "setSVMC_Z_9" AND NOT "setAlarm_Moment_Z_9",   // "VLV02"
                 SVMO := "setSVMO_Z_9" AND NOT "setAlarm_Moment_Z_9",
                 CLSD := "inputZamkniętaZ_9",
                 OPND := "inputOtwartaZ_9",
                 REMT := "inputREM_Zasuwy",
                 KT1 := "dbTimersForDrivers".TimerZ8.PT,
                 CLSE := "CMD_Close_Z_9",
                 OPEN := "CMD_Open_Z_9",
                 WIZ := %DB10.DBB22,
                 STAT := %DB10.DBB23,
                 TMR1 := "dbTimersForDrivers".TimerZ9);
END_REGION
END_FUNCTION

FUNCTION_BLOCK "VLV02_POSITION"   // FB6, LAD
TITLE = Valve driver 02
{ S7_Optimized_Access := 'FALSE' }
AUTHOR : RTecmer
VERSION : 0.2
// Driver 0-100% position drives
// Slowo STATUSU Napedu
// STAT - Prawy Byte
// WIZ  - Lewy Byte
//  
//   -STAT wektor stanu zaworu
//     -bit 0- alarm                                  (sygnal do SCADA)
//     -bit 1- zawor otwarty                    (sygnal do SCADA)
//     -bit 2-sterowanie zdal=1 loc=0 (sygnal do SCADA)
//     -bit 3- zawor zamkniety               (sygnal do SCADA)
//     -bit 4-otwieranie reczne              (sygnal z SCADA)
//     -bit 5-zamykanie reczne              (sygnal z SCADA)
//     -bit 6-alarm reset                        (sygnal z SCADA
//     -bit 8-auto= 1man=0                  (sygnal z SCADA)
//   -SUPV 
//   -CLSD zawor zamkniety                    - wejscie
//   -OPND zawor otwarty                        - wejscie
//   -REMT sterowanie zdal=1 loc=0      - wejscie
//   -OPEN otwarcie                                  - wyjscie
//   -CLSE zamkniecie                              - wyjscie
//   - TIM1 czas otwierania  
//   - TIM2 czas zamykania
// stored: AutoNumber false, IsIECCheckEnabled false, SetENOAutomatically false, UDAEnableTagReadback false
   VAR_INPUT
      SetOpen_Percent { ExternalAccessible := 'False'; ExternalVisible := 'False'; ExternalWritable := 'False'} : Word;   // Zadany procent otwarcia
      VectorOut { ExternalAccessible := 'False'; ExternalVisible := 'False'; ExternalWritable := 'False'} : Word;   // Wektor otwarcia z nadajnika
      CLSD : Bool;   // Zamknięta
      OPND : Bool;   // Otwarta
      REMT : Bool;   // Sterowanie zdalne =1, remontowe=0
   END_VAR
   VAR_IN_OUT
      CLSE { ExternalAccessible := 'False'; ExternalVisible := 'False'; ExternalWritable := 'False'} : Bool;   // Wyjście zamykanie
      OPEN { ExternalAccessible := 'False'; ExternalVisible := 'False'; ExternalWritable := 'False'} : Bool;   // Wyjście Otwieranie
      WIZ : Byte;   // Wektor SCADA
      STAT : Byte;   // Wektor statusu napędu
      TMR1 : IEC_TIMER;   // Timer
   END_VAR
   VAR_TEMP
      SVMC : Bool;   // Automat na zamykanie
      SVMO : Bool;   // Automat na otwieranie
      man_Close : Bool;   // znacznik zamykania w trymie manual
      man_Open : Bool;   // znacznik otwierania w trybie manual
      instDiffOpen : Real;   // róznica kąta otwarcia zasuwy
      SP_Real : Real;   // Zadana wartość po konwersji
      PV_Real : Real;   // Vektor położeia po konwerski
      Diff_Real : Real;   // różnica po konwersji
      tmpError_Open : Bool;   // pomocniczy znacznik kontroli czasu jazdy na otwieranie
      tmpError_Close : Bool;   // pomocniczy znacznik kontroli czasu jazdy na zamykanie
   END_VAR
BEGIN

REGION Network 1
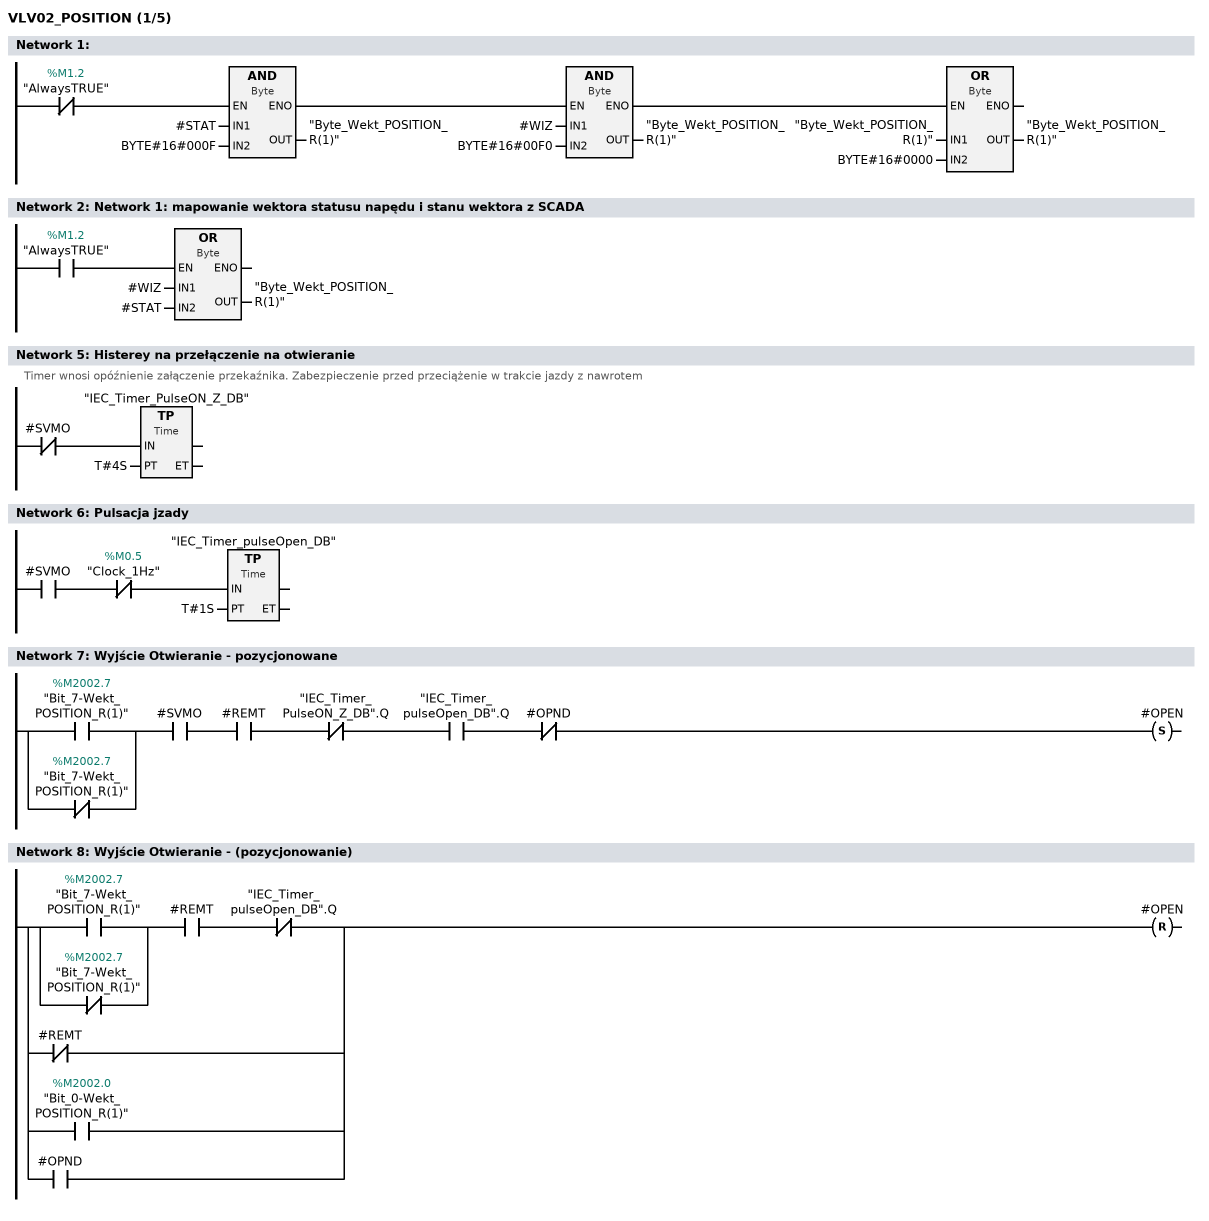
   IF NOT "AlwaysTRUE" THEN
       "Byte_Wekt_POSITION_R(1)" := #STAT AND BYTE#16#000F;
       "Byte_Wekt_POSITION_R(1)" := #WIZ AND BYTE#16#00F0;
       "Byte_Wekt_POSITION_R(1)" := "Byte_Wekt_POSITION_R(1)" OR BYTE#16#0000;
   END_IF;
END_REGION

REGION Network 2: Network 1: mapowanie wektora statusu napędu i stanu wektora z SCADA
   IF "AlwaysTRUE" THEN "Byte_Wekt_POSITION_R(1)" := #WIZ OR #STAT; END_IF;
END_REGION

REGION Network 3 (SCL): wyliczenie różnicy położenia
   //wyliczenie różnicy położenia
   REGION Konwersja zmiennych 
     // Konwersja do Real
     #SP_Real := INT_TO_REAL(#SetOpen_Percent);
     #PV_Real := INT_TO_REAL(#VectorOut);

   END_REGION

   #Diff_Real := (#SP_Real - #PV_Real);
   #instDiffOpen := #Diff_Real;
END_REGION

REGION Network 4 (SCL): Wyznaczenie wektora i jazda na otwierane


   //Strowanie na otwieranie 
   IF #REMT AND "isGotowość_Z_10" THEN
     // Porównaj wartość różnicy do 1
     IF #instDiffOpen > 1.0 AND (#OPND = FALSE )AND (#REMT = TRUE) THEN
       // ustaw znacznik automatyczne otwieranie
       #SVMO := TRUE;
       // znacznik do kontroli czasu 
       #tmpError_Open := TRUE;
     ELSE
       #SVMO := FALSE;
       #tmpError_Open:= FALSE
       ;
     END_IF;

     ;
   END_IF;
END_REGION

REGION Network 5: Histerey na przełączenie na otwieranie
   // Timer wnosi opóźnienie załączenie przekaźnika. Zabezpieczenie przed przeciążenie w trakcie jazdy z nawrotem
   RUNG wire#powerrail
      I_Contact( #SVMO )
      { S7_Templates := "time_type := Time" } "IEC_Timer_PulseON_Z_DB".TP(pt := T#4S, et =>)
   END_RUNG
   // the same network as SCL:
   "IEC_Timer_PulseON_Z_DB".TP(IN := NOT #SVMO, PT := T#4S);
END_REGION

REGION Network 6: Pulsacja jzady
   RUNG wire#powerrail
      Contact( #SVMO )
      I_Contact( "Clock_1Hz" )
      { S7_Templates := "time_type := Time" } "IEC_Timer_pulseOpen_DB".TP(pt := T#1S, et =>)
   END_RUNG
   // the same network as SCL:
   "IEC_Timer_pulseOpen_DB".TP(IN := #SVMO AND NOT "Clock_1Hz", PT := T#1S);
END_REGION

REGION Network 7: Wyjście Otwieranie - pozycjonowane
   RUNG wire#powerrail
      Contact( "Bit_7-Wekt_POSITION_R(1)" )
      wire#w1
      Contact( #SVMO )
      Contact( #REMT )
      I_Contact( "IEC_Timer_PulseON_Z_DB".Q )
      Contact( "IEC_Timer_pulseOpen_DB".Q )
      I_Contact( #OPND )
      S_Coil( #OPEN )
   END_RUNG
   RUNG wire#powerrail
      I_Contact( "Bit_7-Wekt_POSITION_R(1)" )
   END_RUNG wire#w1
   // the same network as SCL:
   IF ("Bit_7-Wekt_POSITION_R(1)" OR NOT "Bit_7-Wekt_POSITION_R(1)") AND #SVMO AND #REMT AND NOT "IEC_Timer_PulseON_Z_DB".Q AND "IEC_Timer_pulseOpen_DB".Q AND NOT #OPND THEN
       #OPEN := TRUE;
   END_IF;
END_REGION

REGION Network 8: Wyjście Otwieranie - (pozycjonowanie)
   RUNG wire#powerrail
      Contact( "Bit_7-Wekt_POSITION_R(1)" )
      wire#w1
      Contact( #REMT )
      I_Contact( "IEC_Timer_pulseOpen_DB".Q )
      wire#w2
      R_Coil( #OPEN )
   END_RUNG
   RUNG wire#powerrail
      I_Contact( "Bit_7-Wekt_POSITION_R(1)" )
   END_RUNG wire#w1
   RUNG wire#powerrail
      I_Contact( #REMT )
   END_RUNG wire#w2
   RUNG wire#powerrail
      Contact( "Bit_0-Wekt_POSITION_R(1)" )
   END_RUNG wire#w2
   RUNG wire#powerrail
      Contact( #OPND )
   END_RUNG wire#w2
   // the same network as SCL:
   IF (("Bit_7-Wekt_POSITION_R(1)" OR NOT "Bit_7-Wekt_POSITION_R(1)") AND #REMT AND NOT "IEC_Timer_pulseOpen_DB".Q) OR NOT #REMT OR "Bit_0-Wekt_POSITION_R(1)" OR #OPND THEN
       #OPEN := FALSE;
   END_IF;
END_REGION

REGION Network 9 (SCL): Wyznaczenie wektora i jazda na zamykanie



   //Strowanie na zamykanie
   IF #REMT AND "isGotowość_Z_10"THEN
     // Porównaj wartość różnicy do 1
     IF #instDiffOpen < -1.0 AND (#CLSD = FALSE) AND (#REMT = TRUE) THEN
       // ustaw znacznik automatyczne zamykanie
       #SVMC := TRUE;
       // znacznik kontroli czasu jazdy
       #tmpError_Close := TRUE;
     ELSE
       #SVMC := FALSE;
       #tmpError_Close:= FALSE
       ;
     END_IF;

     ;
   END_IF;
END_REGION

REGION Network 10: Histerez na przełączenie na zamykanie
   // Timer wnosi opóźnienie załączenie przekaźnika. Zabezpieczenie przed przeciążenie w trakcie jazdy z nawrotem
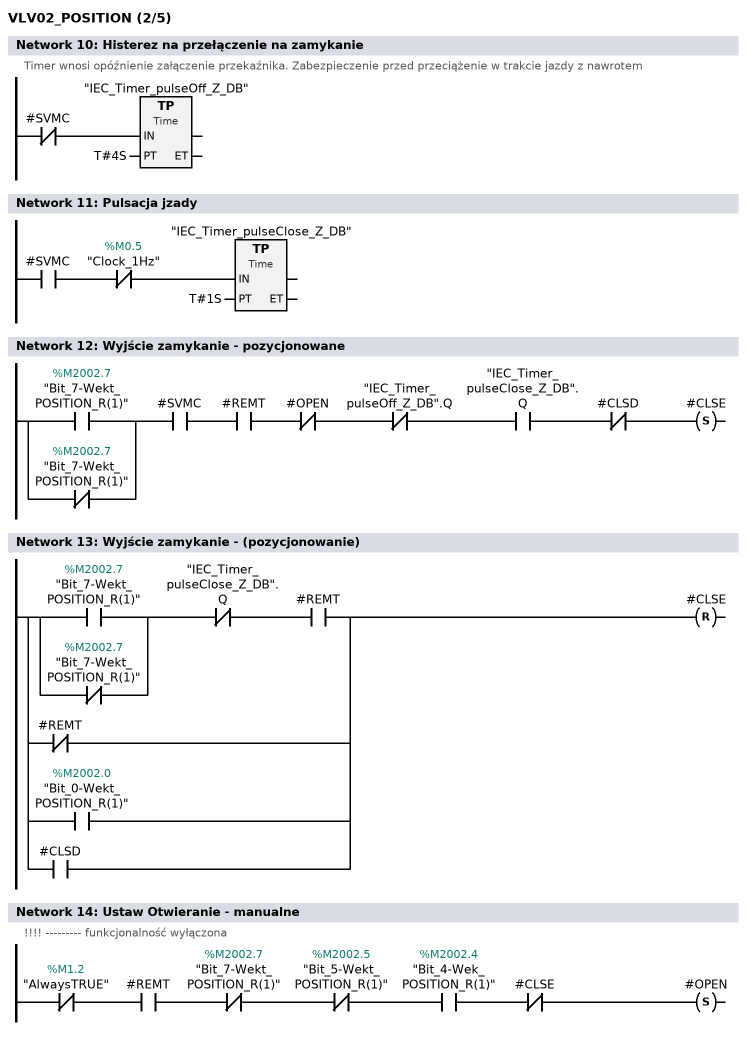
   RUNG wire#powerrail
      I_Contact( #SVMC )
      { S7_Templates := "time_type := Time" } "IEC_Timer_pulseOff_Z_DB".TP(pt := T#4S, et =>)
   END_RUNG
   // the same network as SCL:
   "IEC_Timer_pulseOff_Z_DB".TP(IN := NOT #SVMC, PT := T#4S);
END_REGION

REGION Network 11: Pulsacja jzady
   RUNG wire#powerrail
      Contact( #SVMC )
      I_Contact( "Clock_1Hz" )
      { S7_Templates := "time_type := Time" } "IEC_Timer_pulseClose_Z_DB".TP(pt := T#1S, et =>)
   END_RUNG
   // the same network as SCL:
   "IEC_Timer_pulseClose_Z_DB".TP(IN := #SVMC AND NOT "Clock_1Hz", PT := T#1S);
END_REGION

REGION Network 12: Wyjście zamykanie - pozycjonowane
   RUNG wire#powerrail
      Contact( "Bit_7-Wekt_POSITION_R(1)" )
      wire#w1
      Contact( #SVMC )
      Contact( #REMT )
      I_Contact( #OPEN )
      I_Contact( "IEC_Timer_pulseOff_Z_DB".Q )
      Contact( "IEC_Timer_pulseClose_Z_DB".Q )
      I_Contact( #CLSD )
      S_Coil( #CLSE )
   END_RUNG
   RUNG wire#powerrail
      I_Contact( "Bit_7-Wekt_POSITION_R(1)" )
   END_RUNG wire#w1
   // the same network as SCL:
   IF ("Bit_7-Wekt_POSITION_R(1)" OR NOT "Bit_7-Wekt_POSITION_R(1)") AND #SVMC AND #REMT AND NOT #OPEN AND NOT "IEC_Timer_pulseOff_Z_DB".Q AND "IEC_Timer_pulseClose_Z_DB".Q AND NOT #CLSD THEN
       #CLSE := TRUE;
   END_IF;
END_REGION

REGION Network 13: Wyjście zamykanie - (pozycjonowanie)
   RUNG wire#powerrail
      Contact( "Bit_7-Wekt_POSITION_R(1)" )
      wire#w1
      I_Contact( "IEC_Timer_pulseClose_Z_DB".Q )
      Contact( #REMT )
      wire#w2
      R_Coil( #CLSE )
   END_RUNG
   RUNG wire#powerrail
      I_Contact( "Bit_7-Wekt_POSITION_R(1)" )
   END_RUNG wire#w1
   RUNG wire#powerrail
      I_Contact( #REMT )
   END_RUNG wire#w2
   RUNG wire#powerrail
      Contact( "Bit_0-Wekt_POSITION_R(1)" )
   END_RUNG wire#w2
   RUNG wire#powerrail
      Contact( #CLSD )
   END_RUNG wire#w2
   // the same network as SCL:
   IF (("Bit_7-Wekt_POSITION_R(1)" OR NOT "Bit_7-Wekt_POSITION_R(1)") AND NOT "IEC_Timer_pulseClose_Z_DB".Q AND #REMT) OR NOT #REMT OR "Bit_0-Wekt_POSITION_R(1)" OR #CLSD THEN
       #CLSE := FALSE;
   END_IF;
END_REGION

REGION Network 14: Ustaw Otwieranie - manualne
   // !!!! --------- funkcjonalność wyłączona
   RUNG wire#powerrail
      I_Contact( "AlwaysTRUE" )
      Contact( #REMT )
      I_Contact( "Bit_7-Wekt_POSITION_R(1)" )
      I_Contact( "Bit_5-Wekt_POSITION_R(1)" )
      Contact( "Bit_4-Wek_POSITION_R(1)" )
      I_Contact( #CLSE )
      S_Coil( #OPEN )
   END_RUNG
   // the same network as SCL:
   IF NOT "AlwaysTRUE" AND #REMT AND NOT "Bit_7-Wekt_POSITION_R(1)" AND NOT "Bit_5-Wekt_POSITION_R(1)" AND "Bit_4-Wek_POSITION_R(1)" AND NOT #CLSE THEN
       #OPEN := TRUE;
   END_IF;
END_REGION

REGION Network 15: Reset Otwieranie
   // dodałem reset gdy wydano rozkaz zamykania
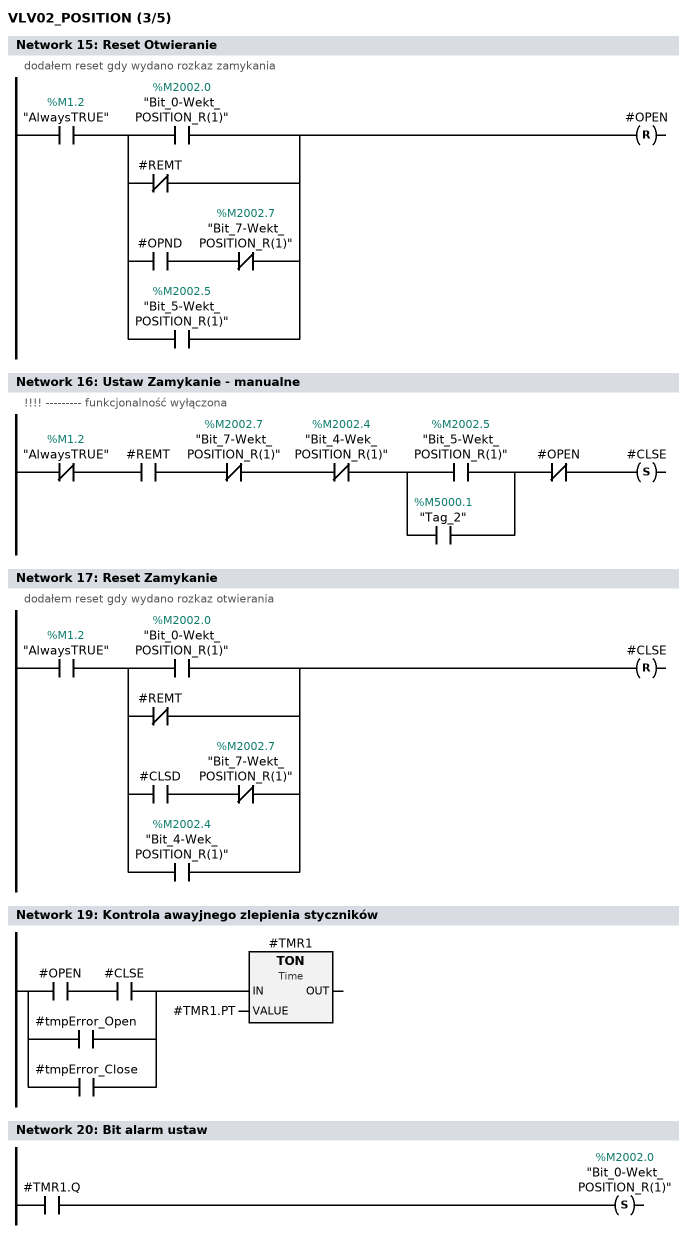
   RUNG wire#powerrail
      Contact( "AlwaysTRUE" )
      wire#w1
      Contact( "Bit_0-Wekt_POSITION_R(1)" )
      wire#w2
      R_Coil( #OPEN )
   END_RUNG
   RUNG wire#w1
      I_Contact( #REMT )
   END_RUNG wire#w2
   RUNG wire#w1
      Contact( #OPND )
      I_Contact( "Bit_7-Wekt_POSITION_R(1)" )
   END_RUNG wire#w2
   RUNG wire#w1
      Contact( "Bit_5-Wekt_POSITION_R(1)" )
   END_RUNG wire#w2
   // the same network as SCL:
   IF "AlwaysTRUE" AND ("Bit_0-Wekt_POSITION_R(1)" OR NOT #REMT OR (#OPND AND NOT "Bit_7-Wekt_POSITION_R(1)") OR "Bit_5-Wekt_POSITION_R(1)") THEN
       #OPEN := FALSE;
   END_IF;
END_REGION

REGION Network 16: Ustaw Zamykanie - manualne
   // !!!! --------- funkcjonalność wyłączona
   RUNG wire#powerrail
      I_Contact( "AlwaysTRUE" )
      Contact( #REMT )
      I_Contact( "Bit_7-Wekt_POSITION_R(1)" )
      I_Contact( "Bit_4-Wek_POSITION_R(1)" )
      wire#w1
      Contact( "Bit_5-Wekt_POSITION_R(1)" )
      wire#w2
      I_Contact( #OPEN )
      S_Coil( #CLSE )
   END_RUNG
   RUNG wire#w1
      Contact( "Tag_2" )
   END_RUNG wire#w2
   // the same network as SCL:
   IF NOT "AlwaysTRUE" AND #REMT AND NOT "Bit_7-Wekt_POSITION_R(1)" AND NOT "Bit_4-Wek_POSITION_R(1)" AND ("Bit_5-Wekt_POSITION_R(1)" OR "Tag_2") AND NOT #OPEN THEN
       #CLSE := TRUE;
   END_IF;
END_REGION

REGION Network 17: Reset Zamykanie
   // dodałem reset gdy wydano rozkaz otwierania
   RUNG wire#powerrail
      Contact( "AlwaysTRUE" )
      wire#w1
      Contact( "Bit_0-Wekt_POSITION_R(1)" )
      wire#w2
      R_Coil( #CLSE )
   END_RUNG
   RUNG wire#w1
      I_Contact( #REMT )
   END_RUNG wire#w2
   RUNG wire#w1
      Contact( #CLSD )
      I_Contact( "Bit_7-Wekt_POSITION_R(1)" )
   END_RUNG wire#w2
   RUNG wire#w1
      Contact( "Bit_4-Wek_POSITION_R(1)" )
   END_RUNG wire#w2
   // the same network as SCL:
   IF "AlwaysTRUE" AND ("Bit_0-Wekt_POSITION_R(1)" OR NOT #REMT OR (#CLSD AND NOT "Bit_7-Wekt_POSITION_R(1)") OR "Bit_4-Wek_POSITION_R(1)") THEN
       #CLSE := FALSE;
   END_IF;
END_REGION

REGION Network 19: Kontrola awayjnego zlepienia styczników
   #TMR1.TON(IN := (#OPEN AND #CLSE) OR #tmpError_Open OR #tmpError_Close, PT := #TMR1.PT);   // TON coil
END_REGION

REGION Network 20: Bit alarm ustaw
   RUNG wire#powerrail
      Contact( #TMR1.Q )
      S_Coil( "Bit_0-Wekt_POSITION_R(1)" )
   END_RUNG
   // the same network as SCL:
   IF #TMR1.Q THEN "Bit_0-Wekt_POSITION_R(1)" := TRUE; END_IF;
END_REGION

REGION Network 21: Kasowanie Bitu alarmu
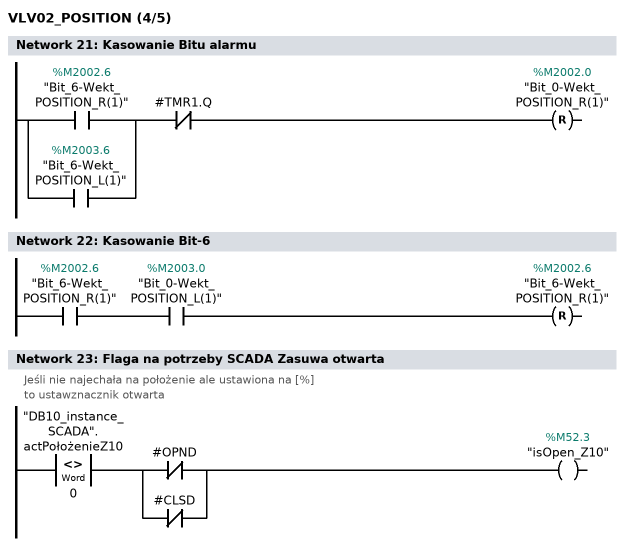
   RUNG wire#powerrail
      Contact( "Bit_6-Wekt_POSITION_R(1)" )
      wire#w1
      I_Contact( #TMR1.Q )
      R_Coil( "Bit_0-Wekt_POSITION_R(1)" )
   END_RUNG
   RUNG wire#powerrail
      Contact( "Bit_6-Wekt_POSITION_L(1)" )
   END_RUNG wire#w1
   // the same network as SCL:
   IF ("Bit_6-Wekt_POSITION_R(1)" OR "Bit_6-Wekt_POSITION_L(1)") AND NOT #TMR1.Q THEN
       "Bit_0-Wekt_POSITION_R(1)" := FALSE;
   END_IF;
END_REGION

REGION Network 22: Kasowanie Bit-6
   RUNG wire#powerrail
      Contact( "Bit_6-Wekt_POSITION_R(1)" )
      Contact( "Bit_0-Wekt_POSITION_L(1)" )
      R_Coil( "Bit_6-Wekt_POSITION_R(1)" )
   END_RUNG
   // the same network as SCL:
   IF "Bit_6-Wekt_POSITION_R(1)" AND "Bit_0-Wekt_POSITION_L(1)" THEN
       "Bit_6-Wekt_POSITION_R(1)" := FALSE;
   END_IF;
END_REGION

REGION Network 23: Flaga na potrzeby SCADA Zasuwa otwarta
   // Jeśli nie najechała na położenie ale ustawiona na [%]
   // to ustawznacznik otwarta
   RUNG wire#powerrail
      { S7_Templates := "SrcType := Word" } NE_Contact(in1 := "DB10_instance_SCADA".actPołożenieZ10, in2 := 0)
      wire#w1
      I_Contact( #OPND )
      wire#w2
      Coil( "isOpen_Z10" )
   END_RUNG
   RUNG wire#w1
      I_Contact( #CLSD )
   END_RUNG wire#w2
   // the same network as SCL:
   "isOpen_Z10" := ("DB10_instance_SCADA".actPołożenieZ10 <> 0) AND (NOT #OPND OR NOT #CLSD);
END_REGION

REGION Network 24: Przepisanie Byte Wektora napędu
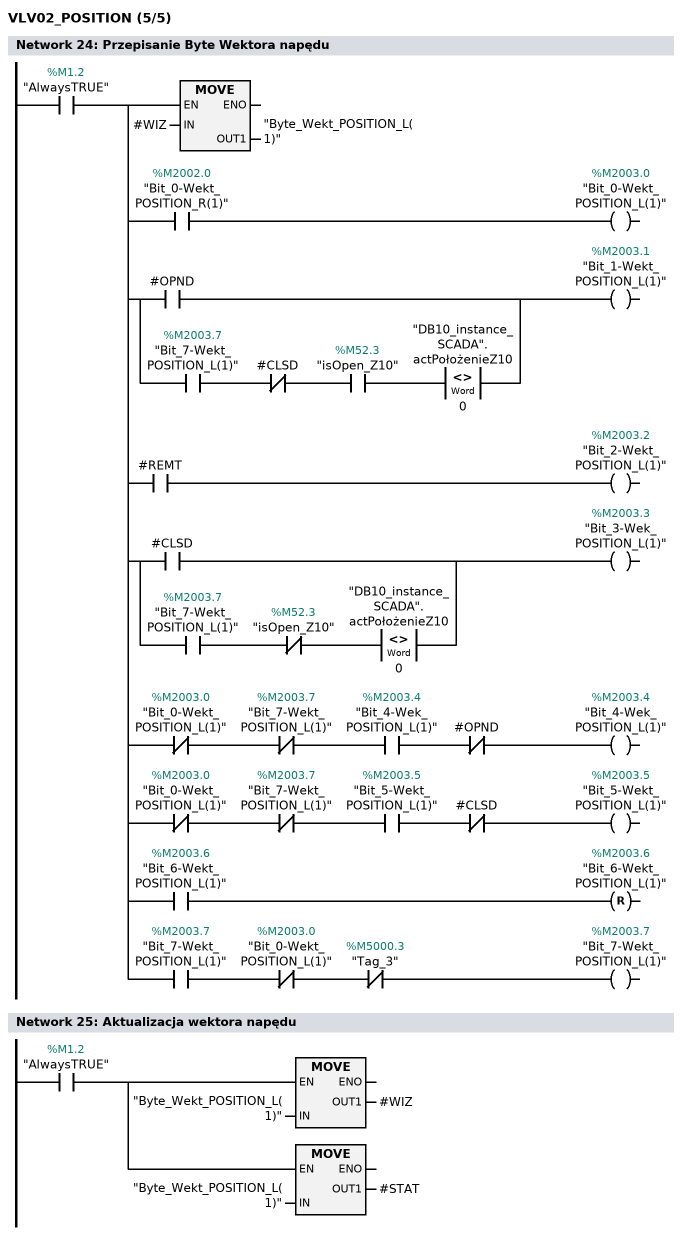
   RUNG wire#powerrail
      Contact( "AlwaysTRUE" )
      wire#w1
      { S7_GenerateENO := "TRUE" } Move(in := #WIZ, out1 => "Byte_Wekt_POSITION_L(1)")
   END_RUNG
   RUNG wire#w1
      Contact( "Bit_0-Wekt_POSITION_R(1)" )
      Coil( "Bit_0-Wekt_POSITION_L(1)" )
   END_RUNG
   RUNG wire#w1
      Contact( #OPND )
      wire#w2
      Coil( "Bit_1-Wekt_POSITION_L(1)" )
   END_RUNG
   RUNG wire#w1
      Contact( "Bit_7-Wekt_POSITION_L(1)" )
      I_Contact( #CLSD )
      Contact( "isOpen_Z10" )
      { S7_Templates := "SrcType := Word" } NE_Contact(in1 := "DB10_instance_SCADA".actPołożenieZ10, in2 := 0)
   END_RUNG wire#w2
   RUNG wire#w1
      Contact( #REMT )
      Coil( "Bit_2-Wekt_POSITION_L(1)" )
   END_RUNG
   RUNG wire#w1
      Contact( #CLSD )
      wire#w3
      Coil( "Bit_3-Wek_POSITION_L(1)" )
   END_RUNG
   RUNG wire#w1
      Contact( "Bit_7-Wekt_POSITION_L(1)" )
      I_Contact( "isOpen_Z10" )
      { S7_Templates := "SrcType := Word" } NE_Contact(in1 := "DB10_instance_SCADA".actPołożenieZ10, in2 := 0)
   END_RUNG wire#w3
   RUNG wire#w1
      I_Contact( "Bit_0-Wekt_POSITION_L(1)" )
      I_Contact( "Bit_7-Wekt_POSITION_L(1)" )
      Contact( "Bit_4-Wek_POSITION_L(1)" )
      I_Contact( #OPND )
      Coil( "Bit_4-Wek_POSITION_L(1)" )
   END_RUNG
   RUNG wire#w1
      I_Contact( "Bit_0-Wekt_POSITION_L(1)" )
      I_Contact( "Bit_7-Wekt_POSITION_L(1)" )
      Contact( "Bit_5-Wekt_POSITION_L(1)" )
      I_Contact( #CLSD )
      Coil( "Bit_5-Wekt_POSITION_L(1)" )
   END_RUNG
   RUNG wire#w1
      Contact( "Bit_6-Wekt_POSITION_L(1)" )
      R_Coil( "Bit_6-Wekt_POSITION_L(1)" )
   END_RUNG
   RUNG wire#w1
      Contact( "Bit_7-Wekt_POSITION_L(1)" )
      I_Contact( "Bit_0-Wekt_POSITION_L(1)" )
      I_Contact( "Tag_3" )
      Coil( "Bit_7-Wekt_POSITION_L(1)" )
   END_RUNG
   // the same network as SCL:
   IF "AlwaysTRUE" THEN "Byte_Wekt_POSITION_L(1)" := #WIZ; END_IF;
   "Bit_0-Wekt_POSITION_L(1)" := "AlwaysTRUE" AND "Bit_0-Wekt_POSITION_R(1)";
   "Bit_1-Wekt_POSITION_L(1)" := "AlwaysTRUE" AND (#OPND OR ("Bit_7-Wekt_POSITION_L(1)" AND NOT #CLSD AND "isOpen_Z10" AND ("DB10_instance_SCADA".actPołożenieZ10 <> 0)));
   "Bit_2-Wekt_POSITION_L(1)" := "AlwaysTRUE" AND #REMT;
   "Bit_3-Wek_POSITION_L(1)" := "AlwaysTRUE" AND (#CLSD OR ("Bit_7-Wekt_POSITION_L(1)" AND NOT "isOpen_Z10" AND ("DB10_instance_SCADA".actPołożenieZ10 <> 0)));
   "Bit_4-Wek_POSITION_L(1)" := "AlwaysTRUE" AND NOT "Bit_0-Wekt_POSITION_L(1)" AND NOT "Bit_7-Wekt_POSITION_L(1)" AND "Bit_4-Wek_POSITION_L(1)" AND NOT #OPND;
   "Bit_5-Wekt_POSITION_L(1)" := "AlwaysTRUE" AND NOT "Bit_0-Wekt_POSITION_L(1)" AND NOT "Bit_7-Wekt_POSITION_L(1)" AND "Bit_5-Wekt_POSITION_L(1)" AND NOT #CLSD;
   IF "AlwaysTRUE" AND "Bit_6-Wekt_POSITION_L(1)" THEN "Bit_6-Wekt_POSITION_L(1)" := FALSE; END_IF;
   "Bit_7-Wekt_POSITION_L(1)" := "AlwaysTRUE" AND "Bit_7-Wekt_POSITION_L(1)" AND NOT "Bit_0-Wekt_POSITION_L(1)" AND NOT "Tag_3";
END_REGION

REGION Network 25: Aktualizacja wektora napędu
   RUNG wire#powerrail
      Contact( "AlwaysTRUE" )
      wire#w1
      { S7_GenerateENO := "TRUE" } Move(in := "Byte_Wekt_POSITION_L(1)", out1 => #WIZ)
   END_RUNG
   RUNG wire#w1
      { S7_GenerateENO := "TRUE" } Move(in := "Byte_Wekt_POSITION_L(1)", out1 => #STAT)
   END_RUNG
   // the same network as SCL:
   IF "AlwaysTRUE" THEN
       #WIZ := "Byte_Wekt_POSITION_L(1)";
       #STAT := "Byte_Wekt_POSITION_L(1)";
   END_IF;
END_REGION
END_FUNCTION_BLOCK

FUNCTION_BLOCK "VLV02"   // FB5, LAD
TITLE = Valve driver 02
{ S7_Optimized_Access := 'FALSE' }
AUTHOR : RTecmer
VERSION : 0.2
// Driver for two-position drives
// Slowo STATUSU Napedu
// STAT - Prawy Byte
// WIZ  - Lewy Byte
//  
//   -STAT wektor stanu zaworu
//     -bit 0- alarm                                  (sygnal do SCADA)
//     -bit 1- zawor otwarty                    (sygnal do SCADA)
//     -bit 2-sterowanie zdal=1 loc=0 (sygnal do SCADA)
//     -bit 3- zawor zamkniety               (sygnal do SCADA)
//     -bit 4-otwieranie reczne              (sygnal z SCADA)
//     -bit 5-zamykanie reczne              (sygnal z SCADA)
//     -bit 6-alarm reset                        (sygnal z SCADA
//     -bit 8-auto= 1man=0                  (sygnal z SCADA)
//   -SUPV 
//   -CLSD zawor zamkniety                    - wejscie
//   -OPND zawor otwarty                        - wejscie
//   -REMT sterowanie zdal=1 loc=0      - wejscie
//   -OPEN otwarcie                                  - wyjscie
//   -CLSE zamkniecie                              - wyjscie
//   - TIM1 czas otwierania  
//   - TIM2 czas zamykania
// stored: AutoNumber true, IsIECCheckEnabled false, SetENOAutomatically false, UDAEnableTagReadback false
   VAR_INPUT
      SVMC : Bool;   // Automat na zamykanie
      SVMO { ExternalVisible := 'False'} : Bool;   // Automat na otwieranie
      CLSD : Bool;   // Zamknięta
      OPND : Bool;   // Otwarta
      REMT : Bool;   // Sterowanie zdalne =1, remontowe=0
      KT1 : Time;   // Czas timera
   END_VAR
   VAR_IN_OUT
      CLSE { ExternalAccessible := 'False'; ExternalVisible := 'False'; ExternalWritable := 'False'} : Bool;   // Wyjście zamykanie
      OPEN { ExternalAccessible := 'False'; ExternalVisible := 'False'; ExternalWritable := 'False'} : Bool;   // Wyjście Otwieranie
      WIZ : Byte;   // Wektor SCADA
      STAT : Byte;   // Wektor statusu napędu
      TMR1 : TON_TIME;
   END_VAR
BEGIN

REGION Network 1
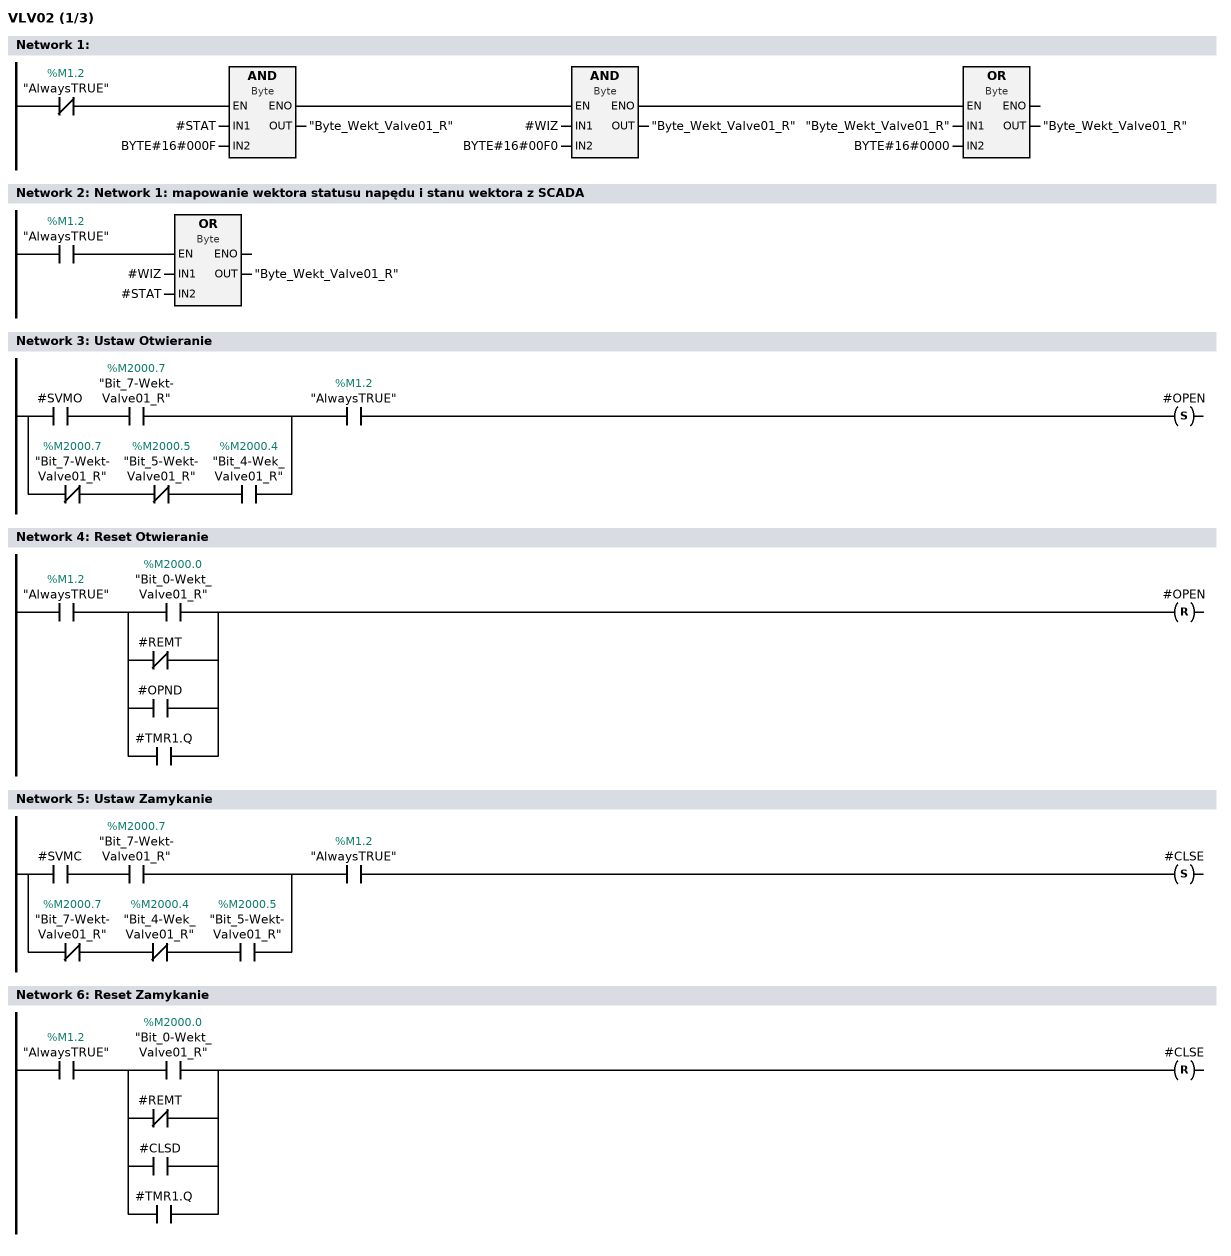
   IF NOT "AlwaysTRUE" THEN
       "Byte_Wekt_Valve01_R" := #STAT AND BYTE#16#000F;
       "Byte_Wekt_Valve01_R" := #WIZ AND BYTE#16#00F0;
       "Byte_Wekt_Valve01_R" := "Byte_Wekt_Valve01_R" OR BYTE#16#0000;
   END_IF;
END_REGION

REGION Network 2: Network 1: mapowanie wektora statusu napędu i stanu wektora z SCADA
   IF "AlwaysTRUE" THEN "Byte_Wekt_Valve01_R" := #WIZ OR #STAT; END_IF;
END_REGION

REGION Network 3: Ustaw Otwieranie
   RUNG wire#powerrail
      Contact( #SVMO )
      Contact( "Bit_7-Wekt-Valve01_R" )
      wire#w1
      Contact( "AlwaysTRUE" )
      S_Coil( #OPEN )
   END_RUNG
   RUNG wire#powerrail
      I_Contact( "Bit_7-Wekt-Valve01_R" )
      I_Contact( "Bit_5-Wekt-Valve01_R" )
      Contact( "Bit_4-Wek_Valve01_R" )
   END_RUNG wire#w1
   // the same network as SCL:
   IF ((#SVMO AND "Bit_7-Wekt-Valve01_R") OR (NOT "Bit_7-Wekt-Valve01_R" AND NOT "Bit_5-Wekt-Valve01_R" AND "Bit_4-Wek_Valve01_R")) AND "AlwaysTRUE" THEN
       #OPEN := TRUE;
   END_IF;
END_REGION

REGION Network 4: Reset Otwieranie
   RUNG wire#powerrail
      Contact( "AlwaysTRUE" )
      wire#w1
      Contact( "Bit_0-Wekt_Valve01_R" )
      wire#w2
      R_Coil( #OPEN )
   END_RUNG
   RUNG wire#w1
      I_Contact( #REMT )
   END_RUNG wire#w2
   RUNG wire#w1
      Contact( #OPND )
   END_RUNG wire#w2
   RUNG wire#w1
      Contact( #TMR1.Q )
   END_RUNG wire#w2
   // the same network as SCL:
   IF "AlwaysTRUE" AND ("Bit_0-Wekt_Valve01_R" OR NOT #REMT OR #OPND OR #TMR1.Q) THEN #OPEN := FALSE; END_IF;
END_REGION

REGION Network 5: Ustaw Zamykanie
   RUNG wire#powerrail
      Contact( #SVMC )
      Contact( "Bit_7-Wekt-Valve01_R" )
      wire#w1
      Contact( "AlwaysTRUE" )
      S_Coil( #CLSE )
   END_RUNG
   RUNG wire#powerrail
      I_Contact( "Bit_7-Wekt-Valve01_R" )
      I_Contact( "Bit_4-Wek_Valve01_R" )
      Contact( "Bit_5-Wekt-Valve01_R" )
   END_RUNG wire#w1
   // the same network as SCL:
   IF ((#SVMC AND "Bit_7-Wekt-Valve01_R") OR (NOT "Bit_7-Wekt-Valve01_R" AND NOT "Bit_4-Wek_Valve01_R" AND "Bit_5-Wekt-Valve01_R")) AND "AlwaysTRUE" THEN
       #CLSE := TRUE;
   END_IF;
END_REGION

REGION Network 6: Reset Zamykanie
   RUNG wire#powerrail
      Contact( "AlwaysTRUE" )
      wire#w1
      Contact( "Bit_0-Wekt_Valve01_R" )
      wire#w2
      R_Coil( #CLSE )
   END_RUNG
   RUNG wire#w1
      I_Contact( #REMT )
   END_RUNG wire#w2
   RUNG wire#w1
      Contact( #CLSD )
   END_RUNG wire#w2
   RUNG wire#w1
      Contact( #TMR1.Q )
   END_RUNG wire#w2
   // the same network as SCL:
   IF "AlwaysTRUE" AND ("Bit_0-Wekt_Valve01_R" OR NOT #REMT OR #CLSD OR #TMR1.Q) THEN #CLSE := FALSE; END_IF;
END_REGION

REGION Network 8: Kontrola czasu jazdy
   // Jeśli wyjście na otwieranie załączone i  brak potwierdzenia otwarcia to załącz  timer na jazdę
   // Jeśli wyjście na zamykanie załączone i j brak potwierdzenia zamknięcia to załącz  timer na jazdę
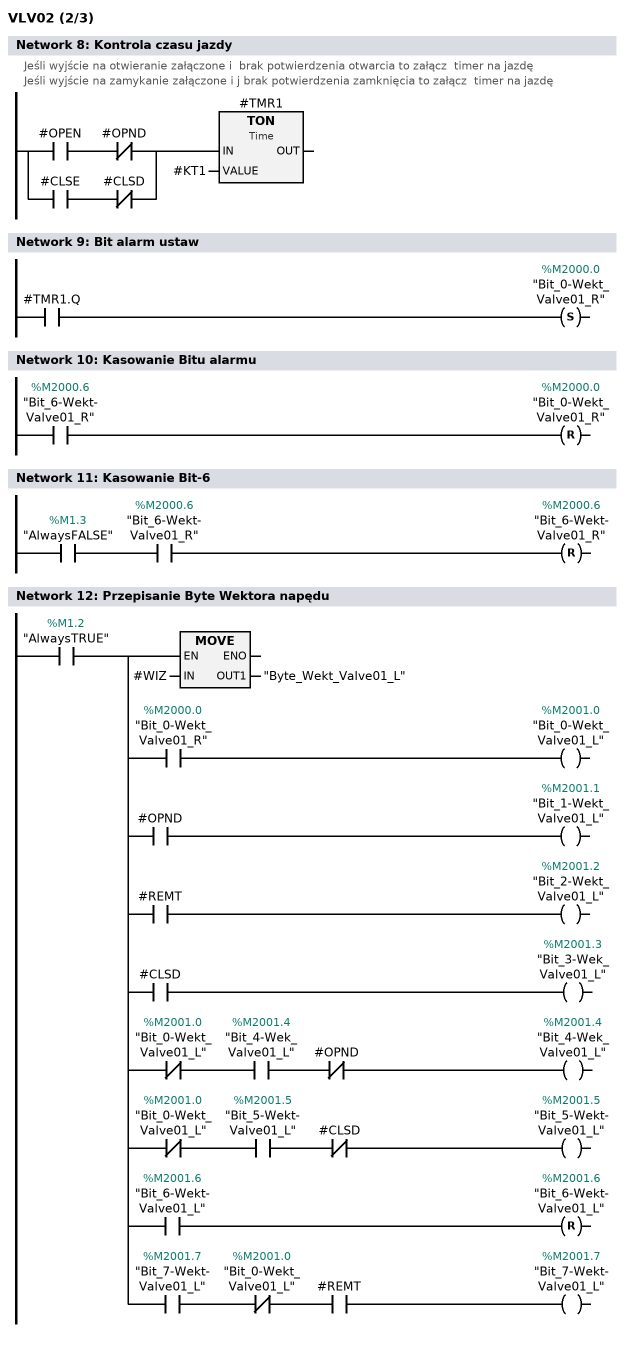
   #TMR1(IN := (#OPEN AND NOT #OPND) OR (#CLSE AND NOT #CLSD), PT := #KT1);   // TON coil
END_REGION

REGION Network 9: Bit alarm ustaw
   RUNG wire#powerrail
      Contact( #TMR1.Q )
      S_Coil( "Bit_0-Wekt_Valve01_R" )
   END_RUNG
   // the same network as SCL:
   IF #TMR1.Q THEN "Bit_0-Wekt_Valve01_R" := TRUE; END_IF;
END_REGION

REGION Network 10: Kasowanie Bitu alarmu
   RUNG wire#powerrail
      Contact( "Bit_6-Wekt-Valve01_R" )
      R_Coil( "Bit_0-Wekt_Valve01_R" )
   END_RUNG
   // the same network as SCL:
   IF "Bit_6-Wekt-Valve01_R" THEN "Bit_0-Wekt_Valve01_R" := FALSE; END_IF;
END_REGION

REGION Network 11: Kasowanie Bit-6
   RUNG wire#powerrail
      Contact( "AlwaysFALSE" )
      Contact( "Bit_6-Wekt-Valve01_R" )
      R_Coil( "Bit_6-Wekt-Valve01_R" )
   END_RUNG
   // the same network as SCL:
   IF "AlwaysFALSE" AND "Bit_6-Wekt-Valve01_R" THEN "Bit_6-Wekt-Valve01_R" := FALSE; END_IF;
END_REGION

REGION Network 12: Przepisanie Byte Wektora napędu
   RUNG wire#powerrail
      Contact( "AlwaysTRUE" )
      wire#w1
      { S7_GenerateENO := "TRUE" } Move(in := #WIZ, out1 => "Byte_Wekt_Valve01_L")
   END_RUNG
   RUNG wire#w1
      Contact( "Bit_0-Wekt_Valve01_R" )
      Coil( "Bit_0-Wekt_Valve01_L" )
   END_RUNG
   RUNG wire#w1
      Contact( #OPND )
      Coil( "Bit_1-Wekt_Valve01_L" )
   END_RUNG
   RUNG wire#w1
      Contact( #REMT )
      Coil( "Bit_2-Wekt_Valve01_L" )
   END_RUNG
   RUNG wire#w1
      Contact( #CLSD )
      Coil( "Bit_3-Wek_Valve01_L" )
   END_RUNG
   RUNG wire#w1
      I_Contact( "Bit_0-Wekt_Valve01_L" )
      Contact( "Bit_4-Wek_Valve01_L" )
      I_Contact( #OPND )
      Coil( "Bit_4-Wek_Valve01_L" )
   END_RUNG
   RUNG wire#w1
      I_Contact( "Bit_0-Wekt_Valve01_L" )
      Contact( "Bit_5-Wekt-Valve01_L" )
      I_Contact( #CLSD )
      Coil( "Bit_5-Wekt-Valve01_L" )
   END_RUNG
   RUNG wire#w1
      Contact( "Bit_6-Wekt-Valve01_L" )
      R_Coil( "Bit_6-Wekt-Valve01_L" )
   END_RUNG
   RUNG wire#w1
      Contact( "Bit_7-Wekt-Valve01_L" )
      I_Contact( "Bit_0-Wekt_Valve01_L" )
      Contact( #REMT )
      Coil( "Bit_7-Wekt-Valve01_L" )
   END_RUNG
   // the same network as SCL:
   IF "AlwaysTRUE" THEN "Byte_Wekt_Valve01_L" := #WIZ; END_IF;
   "Bit_0-Wekt_Valve01_L" := "AlwaysTRUE" AND "Bit_0-Wekt_Valve01_R";
   "Bit_1-Wekt_Valve01_L" := "AlwaysTRUE" AND #OPND;
   "Bit_2-Wekt_Valve01_L" := "AlwaysTRUE" AND #REMT;
   "Bit_3-Wek_Valve01_L" := "AlwaysTRUE" AND #CLSD;
   "Bit_4-Wek_Valve01_L" := "AlwaysTRUE" AND NOT "Bit_0-Wekt_Valve01_L" AND "Bit_4-Wek_Valve01_L" AND NOT #OPND;
   "Bit_5-Wekt-Valve01_L" := "AlwaysTRUE" AND NOT "Bit_0-Wekt_Valve01_L" AND "Bit_5-Wekt-Valve01_L" AND NOT #CLSD;
   IF "AlwaysTRUE" AND "Bit_6-Wekt-Valve01_L" THEN "Bit_6-Wekt-Valve01_L" := FALSE; END_IF;
   "Bit_7-Wekt-Valve01_L" := "AlwaysTRUE" AND "Bit_7-Wekt-Valve01_L" AND NOT "Bit_0-Wekt_Valve01_L" AND #REMT;
END_REGION

REGION Network 13: Aktualizacja wektora napędu
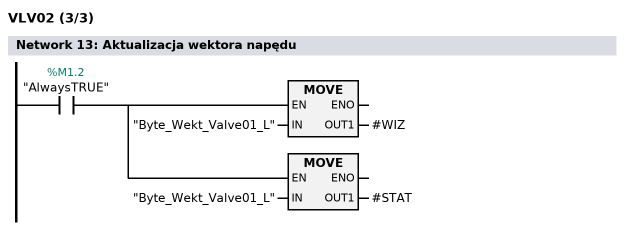
   RUNG wire#powerrail
      Contact( "AlwaysTRUE" )
      wire#w1
      { S7_GenerateENO := "TRUE" } Move(in := "Byte_Wekt_Valve01_L", out1 => #WIZ)
   END_RUNG
   RUNG wire#w1
      { S7_GenerateENO := "TRUE" } Move(in := "Byte_Wekt_Valve01_L", out1 => #STAT)
   END_RUNG
   // the same network as SCL:
   IF "AlwaysTRUE" THEN
       #WIZ := "Byte_Wekt_Valve01_L";
       #STAT := "Byte_Wekt_Valve01_L";
   END_IF;
END_REGION
END_FUNCTION_BLOCK

FUNCTION "D_QUT" : Void
TITLE = Przekazanie wartości 
{ S7_Optimized_Access := 'TRUE' }
AUTHOR : rtecmer
VERSION : 0.1
//Przekazanie wartościna na wyjście cyfrowe (sterowanie wyjściem)

BEGIN
	(*
	//=============================================================================
	//(JZWiK S.A Radosław Tecmer)
	//(c)Copyright (2021) All Rights Reserved
	//-----------------------------------------------------------------------------
	//Testowane z:   (system docelowy z  FW 4.2)
	//Pakiet inżynierski:   TIA Portal (V14 Sp1 Update 9)
	//Ograniczenia:  ( - )
	//Wymagania:  (minimalne S7-1200 CPU 1214 FW 3.2 .)
	//Funkcjonalnośc: (Sterowanie wyjścieami cyfrowymi )
	//-----------------------------------------------------------------------------
	//Zmainy wprowadzone:
	//Wersja  Data       Osoba wprowadzająca zmiany - ekspert
	//01.00.00 28.01.2022 (Tecmer Radosław - twórca) Pieresza wersja 01.00.00
	//=============================================================================
	*)
	
	
	REGION Z10
	  // przekazanie wartości na wyjście
	  "Q2.5":="CMD_Open_Z_10" ;
	  "Q2.6":="CMD_Close_Z_10" ;
	  IF "CMD_Awaria_Z_10" AND "Clock_2Hz" THEN
	    // Sygnalizacja awarii mruganie
	    "Q2.7" := TRUE;
	  ELSE
	    "Q2.7" := FALSE;
	    ;
	  END_IF;
	  
	END_REGION
	
	REGION Z1
	  // przekazanie wartości na wyjście
	  "Q0.3" := "CMD_Open_Z_1";
	  "Q0.4" := "CMD_Close_Z_1";
	  IF "CMD_Awaria_Z_1" AND "Clock_2Hz" THEN
	    // Sygnalizacja awarii mruganie
	    "Q0.5" := TRUE;
	  ELSE
	    "Q0.5" := FALSE;
	    ;
	  END_IF;
	  
	END_REGION
	
	REGION Z2
	  // przekazanie wartości na wyjście
	  "Q3.0" := "CMD_Open_Z_2";
	  "Q3.1" := "CMD_Close_Z_2";
	  IF "CMD_Awaria_Z_2" AND "Clock_2Hz" THEN
	    // Sygnalizacja awarii mruganie
	    "Q3.2" := TRUE;
	  ELSE
	    "Q3.2" := FALSE;
	    ;
	  END_IF;
	  
	END_REGION
	
	REGION Z3
	  // przekazanie wartości na wyjście
	  "Q0.6" := "CMD_Open_Z_3";
	  "Q0.7" := "CMD_Close_Z_3";
	  IF "CMD_Awaria_Z_3" AND "Clock_2Hz" THEN
	    // Sygnalizacja awarii mruganie
	    "Q1.0" := TRUE;
	  ELSE
	    "Q1.0" := FALSE;
	    ;
	  END_IF;
	 
	END_REGION
	
	REGION Z4
	  // przekazanie wartości na wyjście
	  "Q3.4" := "CMD_Open_Z_4";
	  "Q3.5" := "CMD_Close_Z_4";
	  IF "CMD_Awaria_Z_4" AND "Clock_2Hz" THEN
	    // Sygnalizacja awarii mruganie
	    "Q3.6" := TRUE;
	  ELSE
	    "Q3.6" := FALSE;
	    ;
	  END_IF;
	  
	END_REGION
	
	REGION Z5
	  // przekazanie wartości na wyjście
	  "Q1.1" := "CMD_Open_Z_5";
	  "Q2.0" := "CMD_Close_Z_5";
	  IF "CMD_Awaria_Z_5" AND "Clock_2Hz" THEN
	    // Sygnalizacja awarii mruganie
	    "Q2.1" := TRUE;
	  ELSE
	    "Q2.1" := FALSE;
	    ;
	  END_IF;
	  
	END_REGION
	
	REGION Z6
	  // przekazanie wartości na wyjście
	  "Q3.7" := "CMD_Open_Z_6";
	  "Q4.0" := "CMD_Close_Z_6";
	  IF "CMD_Awaria_Z_6" AND "Clock_2Hz" THEN
	    // Sygnalizacja awarii mruganie
	    "Q4.1" := TRUE;
	  ELSE
	    "Q4.1" := FALSE;
	    ;
	  END_IF;
	  
	END_REGION
	
	REGION Z7
	  // przekazanie wartości na wyjście
	  "Q2.2" := "CMD_Open_Z_7";
	  "Q2.3" := "CMD_Close_Z_7";
	  IF "CMD_Awaria_Z_7" AND "Clock_2Hz" THEN
	    // Sygnalizacja awarii mruganie
	    "Q2.4" := TRUE;
	  ELSE
	    "Q2.4" := FALSE;
	    ;
	  END_IF;
	  
	END_REGION
	
	REGION Z8
	  // przekazanie wartości na wyjście
	  "Q4.2" := "CMD_Open_Z_8";
	  "Q4.3" := "CMD_Close_Z_8";
	  IF "CMD_Awaria_Z_8" AND "Clock_2Hz" THEN
	    // Sygnalizacja awarii mruganie
	    "Q4.4" := TRUE;
	  ELSE
	    "Q4.4" := FALSE;
	    ;
	  END_IF;
	  
	END_REGION
	
	REGION Z9
	  // przekazanie wartości na wyjście
	  "Q0.0" := "CMD_Open_Z_9";
	  "Q0.1" := "CMD_Close_Z_9";
	  IF "CMD_Awaria_Z_9" AND "Clock_2Hz" THEN
	    // Sygnalizacja awarii mruganie
	    "Q0.2" := TRUE;
	  ELSE
	    "Q0.2" := FALSE;
	    ;
	  END_IF;
	  
	END_REGION
	
	
	
	
	
	
	
	
	
	
	
	
	
	
	
END_FUNCTION

FUNCTION_BLOCK "Client_ModbusTCP_read_control"   // FB1, LAD
TITLE = Pobieranie parametrów sterowania
{ S7_Optimized_Access := 'TRUE' }
AUTHOR : rtecmer
VERSION : 0.1
// funkcja pobiera z servera dane przekazywanie z PLC 1 do kontroli systemu
// stored: AutoNumber true, IsIECCheckEnabled false, IsRetainMemResEnabled false, MemoryReserve 250, SetENOAutomatically false, UDAEnableTagReadback false
   VAR_IN_OUT
      modbustcp_przetwarzanie_In : Bool;
      modbustcp_przetwarzanie_out : Bool;
   END_VAR
   VAR_TEMP   // added for the SCL form of the ladder/FBD networks
      _w1 : Bool;
      _w2 : Bool;
   END_VAR
BEGIN

REGION Network 1: Inicjacja modbus po błędzie i restarcie
END_REGION

REGION Network 2
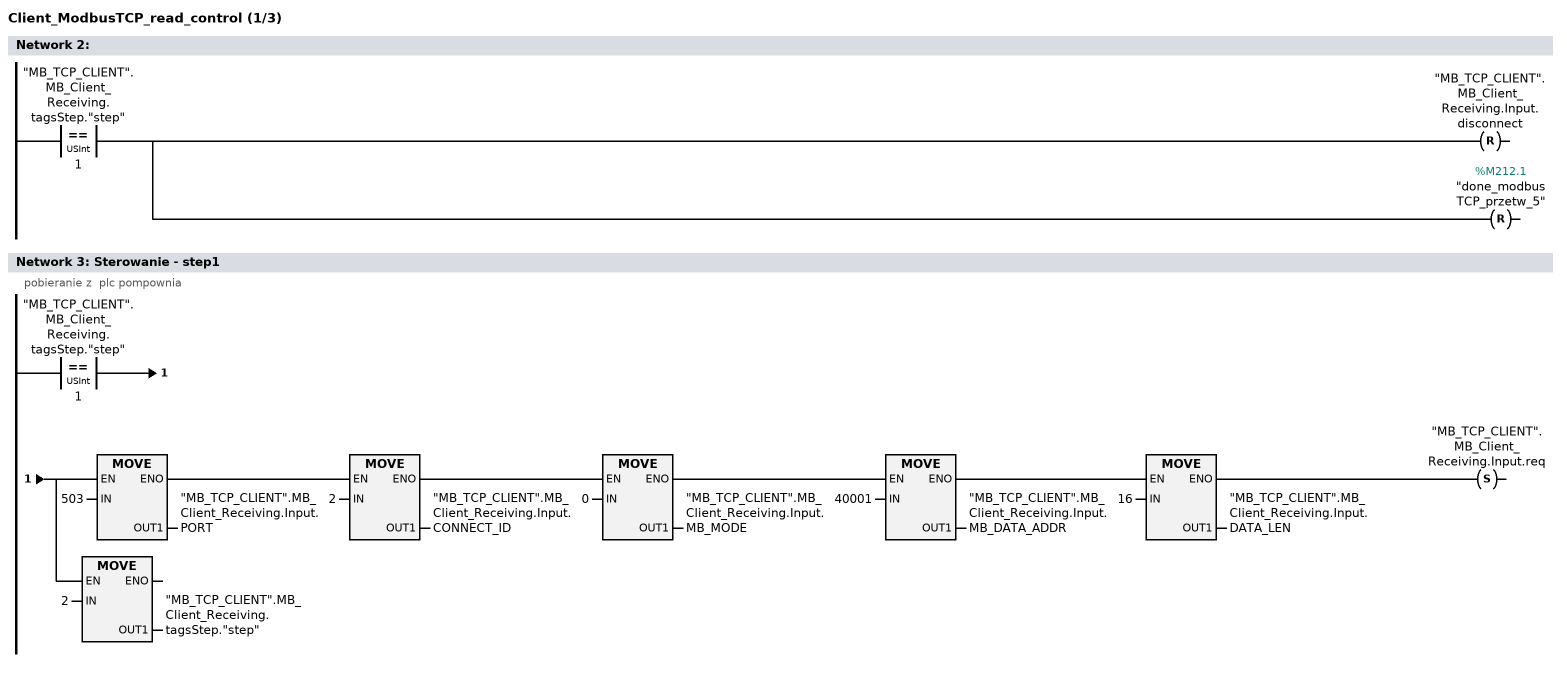
   RUNG wire#powerrail
      { S7_Templates := "SrcType := USInt" } EQ_Contact(in1 := "MB_TCP_CLIENT".MB_Client_Receiving.tagsStep."step", in2 := 1)
      wire#w1
      R_Coil( "MB_TCP_CLIENT".MB_Client_Receiving.Input.disconnect )
   END_RUNG
   RUNG wire#w1
      R_Coil( "done_modbusTCP_przetw_5" )
   END_RUNG
   // the same network as SCL:
   IF "MB_TCP_CLIENT".MB_Client_Receiving.tagsStep."step" = 1 THEN
       "MB_TCP_CLIENT".MB_Client_Receiving.Input.disconnect := FALSE;
       "done_modbusTCP_przetw_5" := FALSE;
   END_IF;
END_REGION

REGION Network 3: Sterowanie - step1
   // pobieranie z  plc pompownia
   RUNG wire#powerrail
      { S7_Templates := "SrcType := USInt" } EQ_Contact(in1 := "MB_TCP_CLIENT".MB_Client_Receiving.tagsStep."step", in2 := 1)
      wire#w1
      { S7_GenerateENO := "TRUE" } Move(in := 503, out1 => "MB_TCP_CLIENT".MB_Client_Receiving.Input.PORT)
      { S7_GenerateENO := "TRUE" } Move(in := 2, out1 => "MB_TCP_CLIENT".MB_Client_Receiving.Input.CONNECT_ID)
      { S7_GenerateENO := "TRUE" } Move(in := 0, out1 => "MB_TCP_CLIENT".MB_Client_Receiving.Input.MB_MODE)
      { S7_GenerateENO := "TRUE" } Move(in := 40001, out1 => "MB_TCP_CLIENT".MB_Client_Receiving.Input.MB_DATA_ADDR)
      { S7_GenerateENO := "TRUE" } Move(in := 16, out1 => "MB_TCP_CLIENT".MB_Client_Receiving.Input.DATA_LEN)
      S_Coil( "MB_TCP_CLIENT".MB_Client_Receiving.Input.req )
   END_RUNG
   RUNG wire#w1
      { S7_GenerateENO := "TRUE" } Move(in := 2, out1 => "MB_TCP_CLIENT".MB_Client_Receiving.tagsStep."step")
   END_RUNG
   // the same network as SCL:
   // ENO of a box is taken as its EN; it also drops when the box reports an error
   IF "MB_TCP_CLIENT".MB_Client_Receiving.tagsStep."step" = 1 THEN
       "MB_TCP_CLIENT".MB_Client_Receiving.Input.PORT := 503;
       "MB_TCP_CLIENT".MB_Client_Receiving.Input.CONNECT_ID := 2;
       "MB_TCP_CLIENT".MB_Client_Receiving.Input.MB_MODE := 0;
       "MB_TCP_CLIENT".MB_Client_Receiving.Input.MB_DATA_ADDR := 40001;
       "MB_TCP_CLIENT".MB_Client_Receiving.Input.DATA_LEN := 16;
       "MB_TCP_CLIENT".MB_Client_Receiving.Input.req := TRUE;
       "MB_TCP_CLIENT".MB_Client_Receiving.tagsStep."step" := 2;
   END_IF;
END_REGION

REGION Network 4: step 2
   // zmienne sterowania
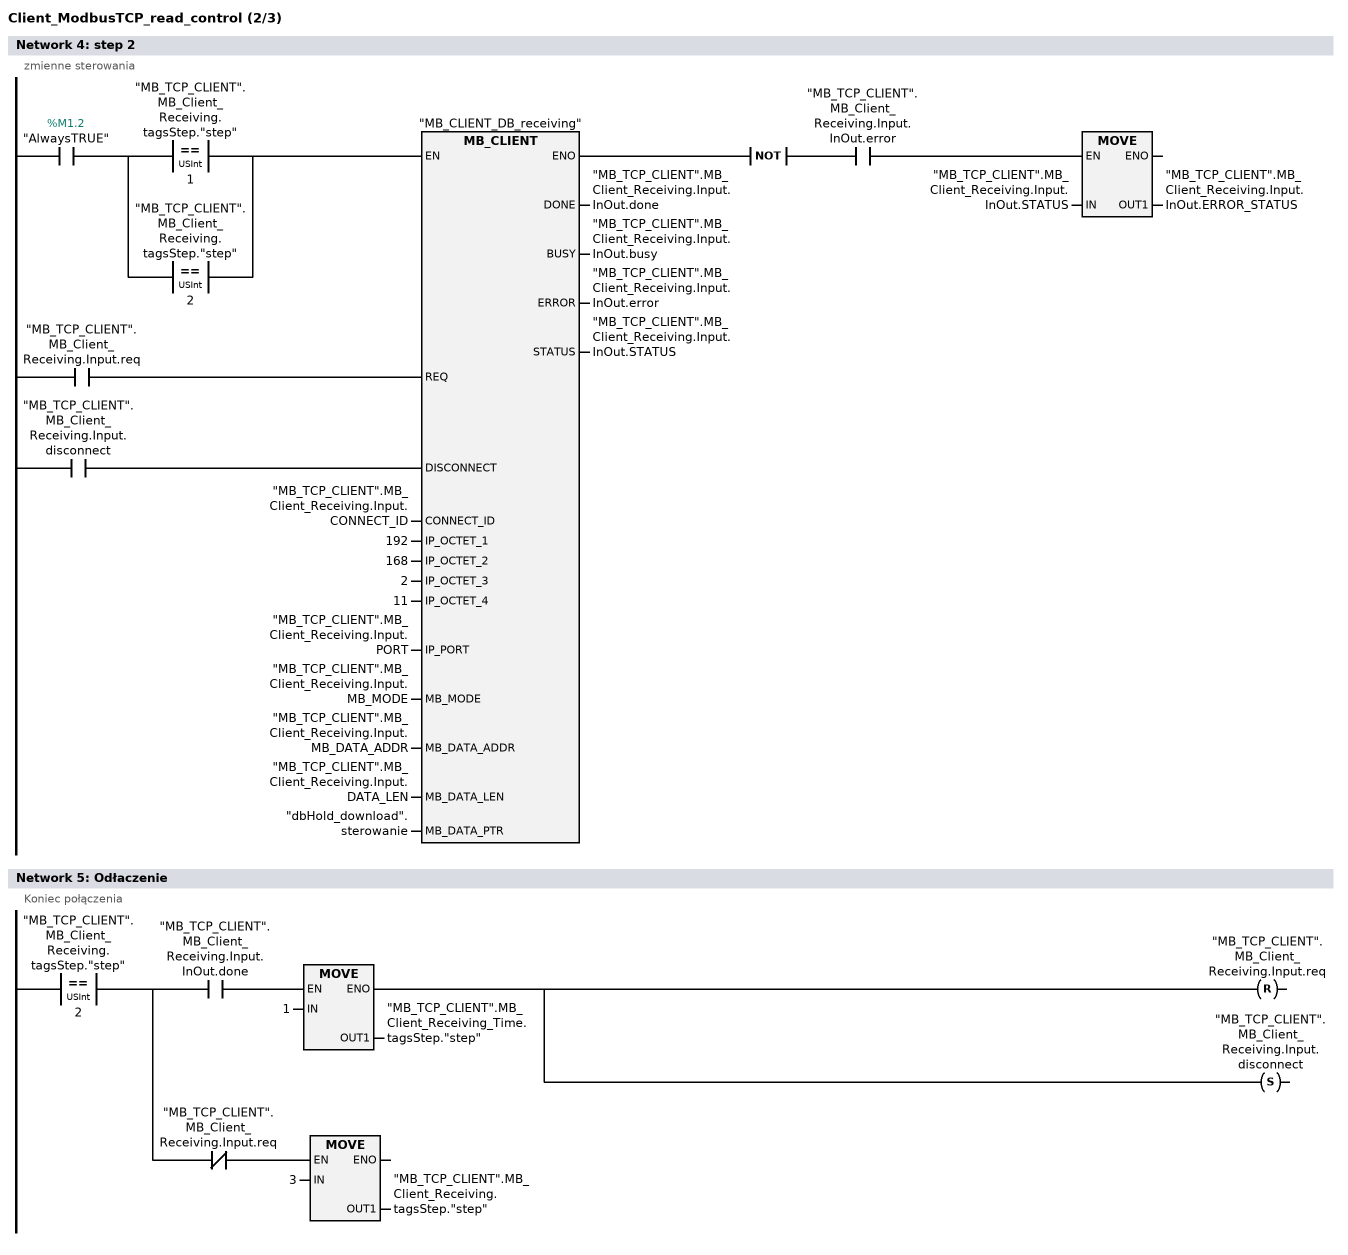
   RUNG wire#powerrail
      Contact( "AlwaysTRUE" )
      wire#w1
      { S7_Templates := "SrcType := USInt" } EQ_Contact(in1 := "MB_TCP_CLIENT".MB_Client_Receiving.tagsStep."step", in2 := 1)
      wire#w2
      { S7_Templates := "[card1200 := 1, card1500 := 0]" } "MB_CLIENT_DB_receiving".MB_CLIENT(REQ := wire#w3, DISCONNECT := wire#w4, CONNECT_ID := "MB_TCP_CLIENT".MB_Client_Receiving.Input.CONNECT_ID, IP_OCTET_1 := 192, IP_OCTET_2 := 168, IP_OCTET_3 := 2, IP_OCTET_4 := 11, IP_PORT := "MB_TCP_CLIENT".MB_Client_Receiving.Input.PORT, MB_MODE := "MB_TCP_CLIENT".MB_Client_Receiving.Input.MB_MODE, MB_DATA_ADDR := "MB_TCP_CLIENT".MB_Client_Receiving.Input.MB_DATA_ADDR, MB_DATA_LEN := "MB_TCP_CLIENT".MB_Client_Receiving.Input.DATA_LEN, MB_DATA_PTR := "dbHold_download".sterowanie, DONE => "MB_TCP_CLIENT".MB_Client_Receiving.Input.InOut.done, BUSY => "MB_TCP_CLIENT".MB_Client_Receiving.Input.InOut.busy, ERROR => "MB_TCP_CLIENT".MB_Client_Receiving.Input.InOut.error, STATUS => "MB_TCP_CLIENT".MB_Client_Receiving.Input.InOut.STATUS)
      Not()
      Contact( "MB_TCP_CLIENT".MB_Client_Receiving.Input.InOut.error )
      Move(in := "MB_TCP_CLIENT".MB_Client_Receiving.Input.InOut.STATUS, out1 => "MB_TCP_CLIENT".MB_Client_Receiving.Input.InOut.ERROR_STATUS)
   END_RUNG
   RUNG wire#w1
      { S7_Templates := "SrcType := USInt" } EQ_Contact(in1 := "MB_TCP_CLIENT".MB_Client_Receiving.tagsStep."step", in2 := 2)
   END_RUNG wire#w2
   RUNG wire#powerrail
      Contact( "MB_TCP_CLIENT".MB_Client_Receiving.Input.req )
   END_RUNG wire#w3
   RUNG wire#powerrail
      Contact( "MB_TCP_CLIENT".MB_Client_Receiving.Input.disconnect )
   END_RUNG wire#w4
   // the same network as SCL:
   #_w1 := "AlwaysTRUE" AND (("MB_TCP_CLIENT".MB_Client_Receiving.tagsStep."step" = 1) OR ("MB_TCP_CLIENT".MB_Client_Receiving.tagsStep."step" = 2));
   "MB_CLIENT_DB_receiving"(EN := #_w1,   // MB_CLIENT
                           REQ := "MB_TCP_CLIENT".MB_Client_Receiving.Input.req,
                           DISCONNECT := "MB_TCP_CLIENT".MB_Client_Receiving.Input.disconnect,
                           CONNECT_ID := "MB_TCP_CLIENT".MB_Client_Receiving.Input.CONNECT_ID,
                           IP_OCTET_1 := 192,
                           IP_OCTET_2 := 168,
                           IP_OCTET_3 := 2,
                           IP_OCTET_4 := 11,
                           IP_PORT := "MB_TCP_CLIENT".MB_Client_Receiving.Input.PORT,
                           MB_MODE := "MB_TCP_CLIENT".MB_Client_Receiving.Input.MB_MODE,
                           MB_DATA_ADDR := "MB_TCP_CLIENT".MB_Client_Receiving.Input.MB_DATA_ADDR,
                           MB_DATA_LEN := "MB_TCP_CLIENT".MB_Client_Receiving.Input.DATA_LEN,
                           MB_DATA_PTR := "dbHold_download".sterowanie,
                           DONE => "MB_TCP_CLIENT".MB_Client_Receiving.Input.InOut.done,
                           BUSY => "MB_TCP_CLIENT".MB_Client_Receiving.Input.InOut.busy,
                           ERROR => "MB_TCP_CLIENT".MB_Client_Receiving.Input.InOut.error,
                           STATUS => "MB_TCP_CLIENT".MB_Client_Receiving.Input.InOut.STATUS,
                           ENO => #_w2);
   IF NOT #_w2 AND "MB_TCP_CLIENT".MB_Client_Receiving.Input.InOut.error THEN
       "MB_TCP_CLIENT".MB_Client_Receiving.Input.InOut.ERROR_STATUS := "MB_TCP_CLIENT".MB_Client_Receiving.Input.InOut.STATUS;
   END_IF;
END_REGION

REGION Network 5: Odłaczenie
   // Koniec połączenia
   RUNG wire#powerrail
      { S7_Templates := "SrcType := USInt" } EQ_Contact(in1 := "MB_TCP_CLIENT".MB_Client_Receiving.tagsStep."step", in2 := 2)
      wire#w1
      Contact( "MB_TCP_CLIENT".MB_Client_Receiving.Input.InOut.done )
      Move(in := 1, out1 => "MB_TCP_CLIENT".MB_Client_Receiving_Time.tagsStep."step")
      wire#w2
      R_Coil( "MB_TCP_CLIENT".MB_Client_Receiving.Input.req )
   END_RUNG
   RUNG wire#w2
      S_Coil( "MB_TCP_CLIENT".MB_Client_Receiving.Input.disconnect )
   END_RUNG
   RUNG wire#w1
      I_Contact( "MB_TCP_CLIENT".MB_Client_Receiving.Input.req )
      Move(in := 3, out1 => "MB_TCP_CLIENT".MB_Client_Receiving.tagsStep."step")
   END_RUNG
   // the same network as SCL:
   #_w1 := "MB_TCP_CLIENT".MB_Client_Receiving.tagsStep."step" = 2;
   IF #_w1 AND "MB_TCP_CLIENT".MB_Client_Receiving.Input.InOut.done THEN
       "MB_TCP_CLIENT".MB_Client_Receiving_Time.tagsStep."step" := 1;
       "MB_TCP_CLIENT".MB_Client_Receiving.Input.req := FALSE;
       "MB_TCP_CLIENT".MB_Client_Receiving.Input.disconnect := TRUE;
   END_IF;
   IF #_w1 AND NOT "MB_TCP_CLIENT".MB_Client_Receiving.Input.req THEN
       "MB_TCP_CLIENT".MB_Client_Receiving.tagsStep."step" := 3;
   END_IF;
END_REGION

REGION Network 6
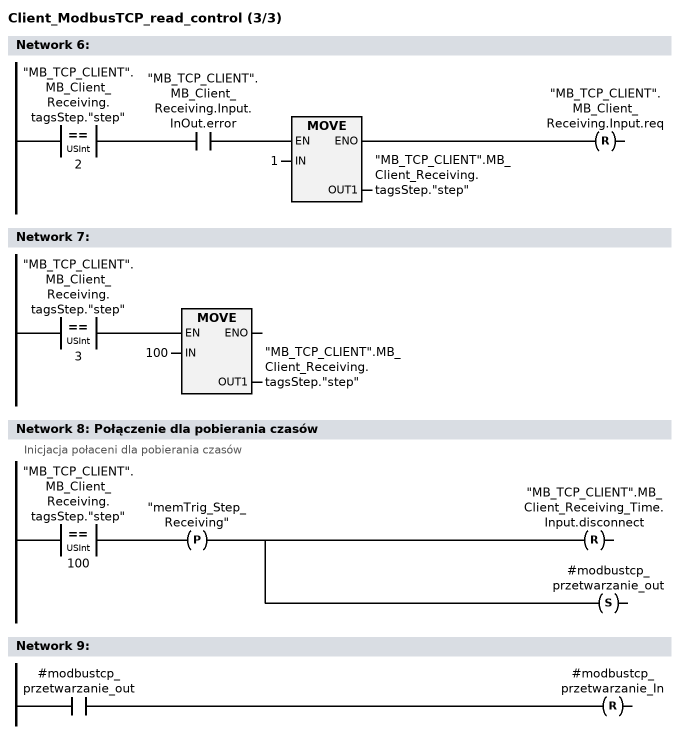
   RUNG wire#powerrail
      { S7_Templates := "SrcType := USInt" } EQ_Contact(in1 := "MB_TCP_CLIENT".MB_Client_Receiving.tagsStep."step", in2 := 2)
      Contact( "MB_TCP_CLIENT".MB_Client_Receiving.Input.InOut.error )
      Move(in := 1, out1 => "MB_TCP_CLIENT".MB_Client_Receiving.tagsStep."step")
      R_Coil( "MB_TCP_CLIENT".MB_Client_Receiving.Input.req )
   END_RUNG
   // the same network as SCL:
   #_w1 := ("MB_TCP_CLIENT".MB_Client_Receiving.tagsStep."step" = 2) AND "MB_TCP_CLIENT".MB_Client_Receiving.Input.InOut.error;
   IF #_w1 THEN
       "MB_TCP_CLIENT".MB_Client_Receiving.tagsStep."step" := 1;
       "MB_TCP_CLIENT".MB_Client_Receiving.Input.req := FALSE;
   END_IF;
END_REGION

REGION Network 7
   RUNG wire#powerrail
      { S7_Templates := "SrcType := USInt" } EQ_Contact(in1 := "MB_TCP_CLIENT".MB_Client_Receiving.tagsStep."step", in2 := 3)
      Move(in := 100, out1 => "MB_TCP_CLIENT".MB_Client_Receiving.tagsStep."step")
   END_RUNG
   // the same network as SCL:
   IF "MB_TCP_CLIENT".MB_Client_Receiving.tagsStep."step" = 3 THEN
       "MB_TCP_CLIENT".MB_Client_Receiving.tagsStep."step" := 100;
   END_IF;
END_REGION

REGION Network 8: Połączenie dla pobierania czasów
   // Inicjacja połaceni dla pobierania czasów
   RUNG wire#powerrail
      { S7_Templates := "SrcType := USInt" } EQ_Contact(in1 := "MB_TCP_CLIENT".MB_Client_Receiving.tagsStep."step", in2 := 100)
      P_Trig( "memTrig_Step_Receiving" )
      wire#w1
      R_Coil( "MB_TCP_CLIENT".MB_Client_Receiving_Time.Input.disconnect )
   END_RUNG
   RUNG wire#w1
      S_Coil( #modbustcp_przetwarzanie_out )
   END_RUNG
   // the same network as SCL:
   #_w1 := "MB_TCP_CLIENT".MB_Client_Receiving.tagsStep."step" = 100;
   #_w2 := #_w1 AND NOT "memTrig_Step_Receiving";   // rising edge
   "memTrig_Step_Receiving" := #_w1;
   IF #_w2 THEN
       "MB_TCP_CLIENT".MB_Client_Receiving_Time.Input.disconnect := FALSE;
       #modbustcp_przetwarzanie_out := TRUE;
   END_IF;
END_REGION

REGION Network 9
   RUNG wire#powerrail
      Contact( #modbustcp_przetwarzanie_out )
      R_Coil( #modbustcp_przetwarzanie_In )
   END_RUNG
   // the same network as SCL:
   IF #modbustcp_przetwarzanie_out THEN #modbustcp_przetwarzanie_In := FALSE; END_IF;
END_REGION
END_FUNCTION_BLOCK

FUNCTION_BLOCK "Client_ModbusTCP_read_DLT"   // FB2, LAD
TITLE = pobieranie czasów
{ S7_Optimized_Access := 'TRUE' }
AUTHOR : rtecmer
VERSION : 0.1
// Funkacja pobiera nastawy czasów
// stored: AutoNumber true, IsIECCheckEnabled false, IsRetainMemResEnabled false, MemoryReserve 250, SetENOAutomatically false, UDAEnableTagReadback false
   VAR_IN_OUT
      modbustcp_przetwarzanie_in : Bool;
      modbustcp_przetwarzanie_out : Bool;
   END_VAR
   VAR_TEMP   // added for the SCL form of the ladder/FBD networks
      _w1 : Bool;
      _w2 : Bool;
   END_VAR
BEGIN

REGION Network 1: Inicjacja modbus po błędzie i restarcie
END_REGION

REGION Network 2
